KUKA KRL program: EPS_2_251806_MH03A_A_20260212042231.src

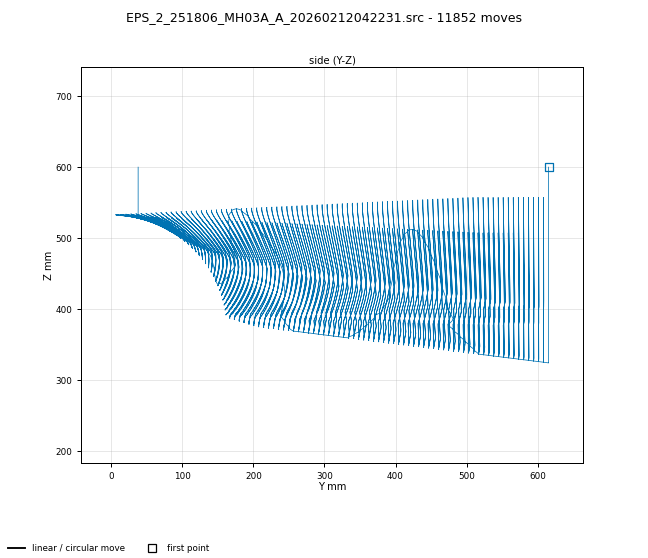
[picture p0: tool path of EPS_2_251806_MH03A_A_20260212042231.src, 11852 of 11854 moves have a stored position in this frame; points joined in program order, loops and branches not executed]
&ACCESS RVP
&REL 4
&COMMENT QRS 19112012
&PARAM EDITMASK = *
DEF PART()
EXT BAS (BAS_COMMAND :IN,REAL :IN )
INT I
BAS (#INITMOV,0 )

;KUKA QRS Post kuka4.cps  Date:22-06-2017 !

File_ID=3011

QRS_PRE_INIT()

;Init var - Until changes are made in qrs_pre_init
Outlet_Square_prg=0
Inlet_1_Square_prg=0
Inlet_2_Square_prg=0
Inlet_3_Square_prg=0
Inlet_4_Square_prg=0
Inlet_5_Square_prg=0

Outlet_1={X 0.000, Y 508.200, Z 408.000, B 0.000, E1 0.000 }
Inlet_1={X 0.000, Y 518.810, Z 382.000, B 0.000, E1 180.000 }
Outlet_1_type=299
Inlet_1_type=251
;QRS#1=Sidecore dimensions
;QRS#2=300-12" PVC SDR 35
;QRS#3=250-10" PVC SDR 35
;QRS#4=
;QRS#5=
;QRS#6=
;QRS#7=
;QRS#8=
;QRS#9=16M PSX
;QRS#10=14M PSX
;QRS#11=
;QRS#12=
;QRS#13=
;QRS#14=
;QRS#15=
;QRS#16=1220x127x838 2,75'
;QRS#17=EPS Height
;QRS#18=557,5
;QRS#19=*
;QRS#20= UPDATED VERSION 22-06-2017
;QRS#21=*
Outlet_Square=0150
Inlet_1_Square=0100
Inlet_2_Square=0
Inlet_3_Square=0
Inlet_4_Square=0
Inlet_5_Square=0
Mill_Square=1
Outlet_Square_Prg=206
Inlet_1_Square_prg=205

QRS_INIT()

$ADVANCE=5

; T1
PTP {E1 173.606,E2 173.606}
PTP {X 0,Y 615.511,A -85,B 0,C 180,E1 173.606,E2 173.606,E3 0,E4 0,E5 0,E6 0}
QRS_SPEED_INIT()
LIN {X 0,Y 615.511,Z 600,A -85,B 0,C 180,E1 173.606,E2 173.606,E3 0,E4 0,E5 0,E6 0} C_VEL
LIN {X 0,Y 615.511,Z 334.496,A -85,B 0,C 180,E1 173.606,E2 173.606} C_VEL
LIN {X 0,Y 615.511,Z 326.325,A -85,B 0,C 180,E1 173.606,E2 173.606} C_VEL
LIN {X 0,Y 615.495,Z 324.325,A -85,B 0,C 180,E1 173.42,E2 173.42} C_VEL
LIN {X 0,Y 615.489,Z 324.313,A -85,B 0,C 180,E1 170.801,E2 170.801} C_VEL
LIN {X 0,Y 615.492,Z 324.321,A -85,B 0,C 180,E1 168.139,E2 168.139} C_VEL
LIN {X 0,Y 615.481,Z 324.317,A -85,B 0,C 180,E1 165.451,E2 165.451} C_VEL
LIN {X 0,Y 615.493,Z 324.313,A -85,B 0,C 180,E1 162.73,E2 162.73} C_VEL
LIN {X 0,Y 615.493,Z 324.325,A -85,B 0,C 180,E1 159.967,E2 159.967} C_VEL
LIN {X 0,Y 615.481,Z 324.316,A -85,B 0,C 180,E1 157.155,E2 157.155} C_VEL
LIN {X 0,Y 615.475,Z 324.319,A -85,B 0,C 180,E1 154.435,E2 154.435} C_VEL
LIN {X 0,Y 615.485,Z 324.315,A -85,B 0,C 180,E1 152.085,E2 152.085} C_VEL
LIN {X 0,Y 615.5,Z 324.325,A -85,B 0,C 180,E1 149.84,E2 149.84} C_VEL
LIN {X 0,Y 615.474,Z 324.317,A -85,B 0,C 180,E1 147.542,E2 147.542} C_VEL
LIN {X 0,Y 615.491,Z 324.317,A -85,B 0,C 180,E1 145.185,E2 145.185} C_VEL
LIN {X 0,Y 615.479,Z 324.32,A -85,B 0,C 180,E1 142.757,E2 142.757} C_VEL
LIN {X 0,Y 615.495,Z 324.321,A -85,B 0,C 180,E1 139.911,E2 139.911} C_VEL
LIN {X 0,Y 615.485,Z 324.315,A -85,B 0,C 180,E1 136.953,E2 136.953} C_VEL
LIN {X 0,Y 615.481,Z 324.315,A -85,B 0,C 180,E1 133.997,E2 133.997} C_VEL
LIN {X 0,Y 615.488,Z 324.324,A -85,B 0,C 180,E1 131.474,E2 131.474} C_VEL
LIN {X 0,Y 615.478,Z 324.315,A -85,B 0,C 180,E1 128.905,E2 128.905} C_VEL
LIN {X 0,Y 615.496,Z 324.364,A -85,B 0,C 180,E1 128.172,E2 128.172} C_VEL
LIN {X 0,Y 615.485,Z 329.475,A -85,B 0,C 180,E1 125.616,E2 125.616} C_VEL
LIN {X 0,Y 615.491,Z 334.286,A -85,B 0,C 180,E1 123.236,E2 123.236} C_VEL
LIN {X 0,Y 615.478,Z 339.068,A -85,B 0,C 180,E1 120.92,E2 120.92} C_VEL
LIN {X 0,Y 615.491,Z 344.306,A -85,B 0,C 180,E1 118.45,E2 118.45} C_VEL
LIN {X 0,Y 615.498,Z 350.554,A -85,B 0,C 180,E1 115.57,E2 115.57} C_VEL
LIN {X 0,Y 615.49,Z 356.619,A -85,B 0,C 180,E1 112.845,E2 112.845} C_VEL
LIN {X 0,Y 615.479,Z 362.996,A -85,B 0,C 180,E1 110.033,E2 110.033} C_VEL
LIN {X 0,Y 615.497,Z 369.367,A -85,B 0,C 180,E1 107.27,E2 107.27} C_VEL
LIN {X 0,Y 615.482,Z 375.745,A -85,B 0,C 180,E1 104.549,E2 104.549} C_VEL
LIN {X 0,Y 615.484,Z 377.068,A -85,B 0,C 180,E1 103.99,E2 103.99} C_VEL
LIN {X 0,Y 615.487,Z 392.156,A -85,B 0,C 180,E1 103.706,E2 103.706} C_VEL
LIN {X 0,Y 615.478,Z 405.741,A -85,B 0,C 180,E1 103.328,E2 103.328} C_VEL
LIN {X 0,Y 615.488,Z 418.034,A -85,B 0,C 180,E1 102.865,E2 102.865} C_VEL
LIN {X 0,Y 615.479,Z 430.302,A -85,B 0,C 180,E1 102.279,E2 102.279} C_VEL
LIN {X 0,Y 615.498,Z 442.906,A -85,B 0,C 180,E1 101.527,E2 101.527} C_VEL
LIN {X 0,Y 615.498,Z 454.072,A -85,B 0,C 180,E1 100.709,E2 100.709} C_VEL
LIN {X 0,Y 615.499,Z 463.697,A -85,B 0,C 180,E1 99.862,E2 99.862} C_VEL
LIN {X 0,Y 615.497,Z 473.147,A -85,B 0,C 180,E1 98.867,E2 98.867} C_VEL
LIN {X 0,Y 615.497,Z 482.137,A -85,B 0,C 180,E1 97.71,E2 97.71} C_VEL
LIN {X 0,Y 615.496,Z 489.382,A -85,B 0,C 180,E1 96.557,E2 96.557} C_VEL
LIN {X 0,Y 615.494,Z 495.887,A -85,B 0,C 180,E1 95.241,E2 95.241} C_VEL
LIN {X 0,Y 615.496,Z 500.757,A -85,B 0,C 180,E1 93.928,E2 93.928} C_VEL
LIN {X 0,Y 615.496,Z 504.154,A -85,B 0,C 180,E1 92.618,E2 92.618} C_VEL
LIN {X 0,Y 615.493,Z 506.174,A -85,B 0,C 180,E1 91.309,E2 91.309} C_VEL
LIN {X 0,Y 615.494,Z 506.884,A -85,B 0,C 180,E1 90,E2 90} C_VEL
LIN {X 0,Y 615.49,Z 506.28,A -85,B 0,C 180,E1 88.691,E2 88.691} C_VEL
LIN {X 0,Y 615.493,Z 504.35,A -85,B 0,C 180,E1 87.382,E2 87.382} C_VEL
LIN {X 0,Y 615.496,Z 501.045,A -85,B 0,C 180,E1 86.071,E2 86.071} C_VEL
LIN {X 0,Y 615.496,Z 496.273,A -85,B 0,C 180,E1 84.759,E2 84.759} C_VEL
LIN {X 0,Y 615.495,Z 489.874,A -85,B 0,C 180,E1 83.443,E2 83.443} C_VEL
LIN {X 0,Y 615.496,Z 482.743,A -85,B 0,C 180,E1 82.289,E2 82.289} C_VEL
LIN {X 0,Y 615.497,Z 475.269,A -85,B 0,C 180,E1 81.298,E2 81.298} C_VEL
LIN {X 0,Y 615.496,Z 466.29,A -85,B 0,C 180,E1 80.304,E2 80.304} C_VEL
LIN {X 0,Y 615.499,Z 455.204,A -85,B 0,C 180,E1 79.291,E2 79.291} C_VEL
LIN {X 0,Y 615.498,Z 444.277,A -85,B 0,C 180,E1 78.473,E2 78.473} C_VEL
LIN {X 0,Y 615.479,Z 431.98,A -85,B 0,C 180,E1 77.721,E2 77.721} C_VEL
LIN {X 0,Y 615.488,Z 420.141,A -85,B 0,C 180,E1 77.134,E2 77.134} C_VEL
LIN {X 0,Y 615.478,Z 407.213,A -85,B 0,C 180,E1 76.63,E2 76.63} C_VEL
LIN {X 0,Y 615.489,Z 394.229,A -85,B 0,C 180,E1 76.252,E2 76.252} C_VEL
LIN {X 0,Y 615.482,Z 379.875,A -85,B 0,C 180,E1 75.972,E2 75.972} C_VEL
LIN {X 0,Y 615.479,Z 377.054,A -85,B 0,C 180,E1 75.914,E2 75.914} C_VEL
LIN {X 0,Y 615.489,Z 371.172,A -85,B 0,C 180,E1 73.413,E2 73.413} C_VEL
LIN {X 0,Y 615.495,Z 364.796,A -85,B 0,C 180,E1 70.662,E2 70.662} C_VEL
LIN {X 0,Y 615.478,Z 358.415,A -85,B 0,C 180,E1 67.863,E2 67.863} C_VEL
LIN {X 0,Y 615.478,Z 352.039,A -85,B 0,C 180,E1 65.008,E2 65.008} C_VEL
LIN {X 0,Y 615.476,Z 347.245,A -85,B 0,C 180,E1 62.822,E2 62.822} C_VEL
LIN {X 0,Y 615.495,Z 341.623,A -85,B 0,C 180,E1 60.205,E2 60.205} C_VEL
LIN {X 0,Y 615.493,Z 336.065,A -85,B 0,C 180,E1 57.542,E2 57.542} C_VEL
LIN {X 0,Y 615.495,Z 331.272,A -85,B 0,C 180,E1 55.185,E2 55.185} C_VEL
LIN {X 0,Y 615.487,Z 326.404,A -85,B 0,C 180,E1 52.757,E2 52.757} C_VEL
LIN {X 0,Y 615.487,Z 324.319,A -85,B 0,C 180,E1 51.619,E2 51.619} C_VEL
LIN {X 0,Y 615.484,Z 324.319,A -85,B 0,C 180,E1 48.906,E2 48.906} C_VEL
LIN {X 0,Y 615.499,Z 324.321,A -85,B 0,C 180,E1 46.756,E2 46.756} C_VEL
LIN {X 0,Y 615.484,Z 324.317,A -85,B 0,C 180,E1 43.996,E2 43.996} C_VEL
LIN {X 0,Y 615.482,Z 324.314,A -85,B 0,C 180,E1 41.093,E2 41.093} C_VEL
LIN {X 0,Y 615.492,Z 324.316,A -85,B 0,C 180,E1 38.904,E2 38.904} C_VEL
LIN {X 0,Y 615.478,Z 324.32,A -85,B 0,C 180,E1 36.426,E2 36.426} C_VEL
LIN {X 0,Y 615.497,Z 324.323,A -85,B 0,C 180,E1 33.535,E2 33.535} C_VEL
LIN {X 0,Y 615.488,Z 324.313,A -85,B 0,C 180,E1 30.92,E2 30.92} C_VEL
LIN {X 0,Y 615.498,Z 324.324,A -85,B 0,C 180,E1 28.451,E2 28.451} C_VEL
LIN {X 0,Y 615.478,Z 324.316,A -85,B 0,C 180,E1 25.716,E2 25.716} C_VEL
LIN {X 0,Y 615.485,Z 324.323,A -85,B 0,C 180,E1 23.557,E2 23.557} C_VEL
LIN {X 0,Y 615.493,Z 324.319,A -85,B 0,C 180,E1 21.432,E2 21.432} C_VEL
LIN {X 0,Y 615.482,Z 324.321,A -85,B 0,C 180,E1 18.601,E2 18.601} C_VEL
LIN {X 0,Y 615.478,Z 324.315,A -85,B 0,C 180,E1 15.906,E2 15.906} C_VEL
LIN {X 0,Y 615.493,Z 324.324,A -85,B 0,C 180,E1 13.201,E2 13.201} C_VEL
LIN {X 0,Y 615.486,Z 324.315,A -85,B 0,C 180,E1 10.527,E2 10.527} C_VEL
LIN {X 0,Y 615.479,Z 324.319,A -85,B 0,C 180,E1 7.876,E2 7.876} C_VEL
LIN {X 0,Y 615.494,Z 324.316,A -85,B 0,C 180,E1 5.241,E2 5.241} C_VEL
LIN {X 0,Y 615.488,Z 324.314,A -85,B 0,C 180,E1 2.618,E2 2.618} C_VEL
LIN {X 0,Y 615.488,Z 324.323,A -85,B 0,C 180,E1 0,E2 0} C_VEL
LIN {X 0,Y 615.488,Z 324.313,A -85,B 0,C 180,E1 -2.618,E2 -2.618} C_VEL
LIN {X 0,Y 615.496,Z 324.324,A -85,B 0,C 180,E1 -5.241,E2 -5.241} C_VEL
LIN {X 0,Y 615.478,Z 324.316,A -85,B 0,C 180,E1 -7.876,E2 -7.876} C_VEL
LIN {X 0,Y 615.486,Z 324.32,A -85,B 0,C 180,E1 -10.527,E2 -10.527} C_VEL
LIN {X 0,Y 615.494,Z 324.316,A -85,B 0,C 180,E1 -13.201,E2 -13.201} C_VEL
LIN {X 0,Y 615.478,Z 324.316,A -85,B 0,C 180,E1 -15.905,E2 -15.905} C_VEL
LIN {X 0,Y 615.493,Z 324.326,A -85,B 0,C 180,E1 -18.646,E2 -18.646} C_VEL
LIN {X 0,Y 615.479,Z 324.317,A -85,B 0,C 180,E1 -21.432,E2 -21.432} C_VEL
LIN {X 0,Y 615.487,Z 324.314,A -85,B 0,C 180,E1 -24.272,E2 -24.272} C_VEL
LIN {X 0,Y 615.49,Z 324.323,A -85,B 0,C 180,E1 -27.177,E2 -27.177} C_VEL
LIN {X 0,Y 615.485,Z 324.315,A -85,B 0,C 180,E1 -29.793,E2 -29.793} C_VEL
LIN {X 0,Y 615.477,Z 324.32,A -85,B 0,C 180,E1 -32.458,E2 -32.458} C_VEL
LIN {X 0,Y 615.491,Z 324.313,A -85,B 0,C 180,E1 -34.815,E2 -34.815} C_VEL
LIN {X 0,Y 615.492,Z 324.323,A -85,B 0,C 180,E1 -37.242,E2 -37.242} C_VEL
LIN {X 0,Y 615.491,Z 324.317,A -85,B 0,C 180,E1 -40.089,E2 -40.089} C_VEL
LIN {X 0,Y 615.483,Z 324.314,A -85,B 0,C 180,E1 -43.046,E2 -43.046} C_VEL
LIN {X 0,Y 615.482,Z 324.317,A -85,B 0,C 180,E1 -46.003,E2 -46.003} C_VEL
LIN {X 0,Y 615.488,Z 324.318,A -85,B 0,C 180,E1 -48.526,E2 -48.526} C_VEL
LIN {X 0,Y 615.478,Z 324.317,A -85,B 0,C 180,E1 -51.094,E2 -51.094} C_VEL
LIN {X 0,Y 615.489,Z 324.318,A -85,B 0,C 180,E1 -53.575,E2 -53.575} C_VEL
LIN {X 0,Y 615.479,Z 324.469,A -85,B 0,C 180,E1 -55.242,E2 -55.242} C_VEL
LIN {X 0,Y 615.492,Z 334.986,A -85,B 0,C 180,E1 -57.992,E2 -57.992} C_VEL
LIN {X 0,Y 615.492,Z 345.267,A -85,B 0,C 180,E1 -60.594,E2 -60.594} C_VEL
LIN {X 0,Y 615.487,Z 356.058,A -85,B 0,C 180,E1 -63.257,E2 -63.257} C_VEL
LIN {X 0,Y 615.478,Z 367.411,A -85,B 0,C 180,E1 -65.994,E2 -65.994} C_VEL
LIN {X 0,Y 615.481,Z 378.295,A -85,B 0,C 180,E1 -68.568,E2 -68.568} C_VEL
LIN {X 0,Y 615.489,Z 390.473,A -85,B 0,C 180,E1 -71.395,E2 -71.395} C_VEL
LIN {X 0,Y 615.488,Z 400.106,A -85,B 0,C 180,E1 -73.601,E2 -73.601} C_VEL
LIN {X 0,Y 615.493,Z 417.365,A -85,B 0,C 180,E1 -73.865,E2 -73.865} C_VEL
LIN {X 0,Y 615.497,Z 432.278,A -85,B 0,C 180,E1 -74.222,E2 -74.222} C_VEL
LIN {X 0,Y 615.478,Z 446.42,A -85,B 0,C 180,E1 -74.689,E2 -74.689} C_VEL
LIN {X 0,Y 615.496,Z 460.354,A -85,B 0,C 180,E1 -75.282,E2 -75.282} C_VEL
LIN {X 0,Y 615.499,Z 473.673,A -85,B 0,C 180,E1 -75.986,E2 -75.986} C_VEL
LIN {X 0,Y 615.498,Z 486.312,A -85,B 0,C 180,E1 -76.799,E2 -76.799} C_VEL
LIN {X 0,Y 615.496,Z 497.291,A -85,B 0,C 180,E1 -77.637,E2 -77.637} C_VEL
LIN {X 0,Y 615.497,Z 508.352,A -85,B 0,C 180,E1 -78.64,E2 -78.64} C_VEL
LIN {X 0,Y 615.496,Z 519.068,A -85,B 0,C 180,E1 -79.806,E2 -79.806} C_VEL
LIN {X 0,Y 615.495,Z 527.987,A -85,B 0,C 180,E1 -80.967,E2 -80.967} C_VEL
LIN {X 0,Y 615.492,Z 535.392,A -85,B 0,C 180,E1 -82.124,E2 -82.124} C_VEL
LIN {X 0,Y 615.491,Z 542.272,A -85,B 0,C 180,E1 -83.443,E2 -83.443} C_VEL
LIN {X 0,Y 615.491,Z 547.666,A -85,B 0,C 180,E1 -84.759,E2 -84.759} C_VEL
LIN {X 0,Y 615.491,Z 551.741,A -85,B 0,C 180,E1 -86.071,E2 -86.071} C_VEL
LIN {X 0,Y 615.496,Z 554.599,A -85,B 0,C 180,E1 -87.382,E2 -87.382} C_VEL
LIN {X 0,Y 615.493,Z 556.306,A -85,B 0,C 180,E1 -88.691,E2 -88.691} C_VEL
LIN {X 0,Y 615.491,Z 556.889,A -85,B 0,C 180,E1 -90,E2 -90} C_VEL
LIN {X 0,Y 615.493,Z 556.307,A -85,B 0,C 180,E1 -91.309,E2 -91.309} C_VEL
LIN {X 0,Y 615.496,Z 554.599,A -85,B 0,C 180,E1 -92.618,E2 -92.618} C_VEL
LIN {X 0,Y 615.491,Z 551.741,A -85,B 0,C 180,E1 -93.928,E2 -93.928} C_VEL
LIN {X 0,Y 615.491,Z 547.666,A -85,B 0,C 180,E1 -95.241,E2 -95.241} C_VEL
LIN {X 0,Y 615.491,Z 542.153,A -85,B 0,C 180,E1 -96.581,E2 -96.581} C_VEL
LIN {X 0,Y 615.492,Z 535.393,A -85,B 0,C 180,E1 -97.876,E2 -97.876} C_VEL
LIN {X 0,Y 615.495,Z 526.809,A -85,B 0,C 180,E1 -99.199,E2 -99.199} C_VEL
LIN {X 0,Y 615.494,Z 517.667,A -85,B 0,C 180,E1 -100.361,E2 -100.361} C_VEL
LIN {X 0,Y 615.497,Z 508.353,A -85,B 0,C 180,E1 -101.36,E2 -101.36} C_VEL
LIN {X 0,Y 615.496,Z 497.292,A -85,B 0,C 180,E1 -102.363,E2 -102.363} C_VEL
LIN {X 0,Y 615.498,Z 485.152,A -85,B 0,C 180,E1 -103.285,E2 -103.285} C_VEL
LIN {X 0,Y 615.498,Z 472.405,A -85,B 0,C 180,E1 -104.09,E2 -104.09} C_VEL
LIN {X 0,Y 615.496,Z 458.609,A -85,B 0,C 180,E1 -104.803,E2 -104.803} C_VEL
LIN {X 0,Y 615.48,Z 444.181,A -85,B 0,C 180,E1 -105.396,E2 -105.396} C_VEL
LIN {X 0,Y 615.496,Z 429.246,A -85,B 0,C 180,E1 -105.863,E2 -105.863} C_VEL
LIN {X 0,Y 615.491,Z 413.842,A -85,B 0,C 180,E1 -106.201,E2 -106.201} C_VEL
LIN {X 0,Y 615.488,Z 400.106,A -85,B 0,C 180,E1 -106.399,E2 -106.399} C_VEL
LIN {X 0,Y 615.484,Z 388.794,A -85,B 0,C 180,E1 -108.992,E2 -108.992} C_VEL
LIN {X 0,Y 615.489,Z 376.797,A -85,B 0,C 180,E1 -111.784,E2 -111.784} C_VEL
LIN {X 0,Y 615.493,Z 364.791,A -85,B 0,C 180,E1 -114.631,E2 -114.631} C_VEL
LIN {X 0,Y 615.494,Z 352.781,A -85,B 0,C 180,E1 -117.545,E2 -117.545} C_VEL
LIN {X 0,Y 615.496,Z 340.758,A -85,B 0,C 180,E1 -120.539,E2 -120.539} C_VEL
LIN {X 0,Y 615.485,Z 330.231,A -85,B 0,C 180,E1 -123.237,E2 -123.237} C_VEL
LIN {X 0,Y 615.478,Z 324.319,A -85,B 0,C 180,E1 -124.816,E2 -124.816} C_VEL
LIN {X 0,Y 615.486,Z 324.315,A -85,B 0,C 180,E1 -127.243,E2 -127.243} C_VEL
LIN {X 0,Y 615.484,Z 324.315,A -85,B 0,C 180,E1 -130.089,E2 -130.089} C_VEL
LIN {X 0,Y 615.498,Z 324.314,A -85,B 0,C 180,E1 -132.353,E2 -132.353} C_VEL
LIN {X 0,Y 615.48,Z 324.316,A -85,B 0,C 180,E1 -135.07,E2 -135.07} C_VEL
LIN {X 0,Y 615.499,Z 324.324,A -85,B 0,C 180,E1 -137.919,E2 -137.919} C_VEL
LIN {X 0,Y 615.491,Z 324.313,A -85,B 0,C 180,E1 -140.25,E2 -140.25} C_VEL
LIN {X 0,Y 615.493,Z 324.322,A -85,B 0,C 180,E1 -143.063,E2 -143.063} C_VEL
LIN {X 0,Y 615.489,Z 324.319,A -85,B 0,C 180,E1 -145.978,E2 -145.978} C_VEL
LIN {X 0,Y 615.484,Z 324.314,A -85,B 0,C 180,E1 -148.915,E2 -148.915} C_VEL
LIN {X 0,Y 615.487,Z 324.321,A -85,B 0,C 180,E1 -151.551,E2 -151.551} C_VEL
LIN {X 0,Y 615.487,Z 324.317,A -85,B 0,C 180,E1 -154.284,E2 -154.284} C_VEL
LIN {X 0,Y 615.481,Z 324.314,A -85,B 0,C 180,E1 -157.155,E2 -157.155} C_VEL
LIN {X 0,Y 615.49,Z 324.32,A -85,B 0,C 180,E1 -159.967,E2 -159.967} C_VEL
LIN {X 0,Y 615.493,Z 324.317,A -85,B 0,C 180,E1 -162.73,E2 -162.73} C_VEL
LIN {X 0,Y 615.482,Z 324.315,A -85,B 0,C 180,E1 -165.451,E2 -165.451} C_VEL
LIN {X 0,Y 615.493,Z 324.326,A -85,B 0,C 180,E1 -168.139,E2 -168.139} C_VEL
LIN {X 0,Y 615.489,Z 324.313,A -85,B 0,C 180,E1 -170.801,E2 -170.801} C_VEL
LIN {X 0,Y 615.496,Z 324.318,A -85,B 0,C 180,E1 -173.444,E2 -173.444} C_VEL
LIN {X 0,Y 615.479,Z 324.318,A -85,B 0,C 180,E1 -176.072,E2 -176.072} C_VEL
LIN {X 0,Y 615.487,Z 324.316,A -85,B 0,C 180,E1 -178.692,E2 -178.692} C_VEL
LIN {X 0,Y 615.487,Z 324.32,A -85,B 0,C 180,E1 -181.309,E2 -181.309} C_VEL
LIN {X 0,Y 615.477,Z 324.316,A -85,B 0,C 180,E1 -183.929,E2 -183.929} C_VEL
LIN {X 0,Y 615.495,Z 324.325,A -85,B 0,C 180,E1 -186.58,E2 -186.58} C_VEL
LIN {X 0,Y 614.815,Z 324.462,A -85,B 0,C 180,E1 -187.126,E2 -187.126} C_VEL
LIN {X 0,Y 611.977,Z 324.88,A -85,B 0,C 180,E1 -188.012,E2 -188.012} C_VEL
LIN {X 0,Y 609.586,Z 325.186,A -85,B 0,C 180,E1 -188.724,E2 -188.724} C_VEL
LIN {X 0,Y 608.552,Z 325.304,A -85,B 0,C 180,E1 -189.274,E2 -189.274} C_VEL
LIN {X 0,Y 608.463,Z 325.315,A -85,B 0,C 180,E1 -189.46,E2 -189.46} C_VEL
LIN {X 0,Y 608.466,Z 325.317,A -85,B 0,C 180,E1 -192,E2 -192} C_VEL
LIN {X 0,Y 608.474,Z 325.316,A -85,B 0,C 180,E1 -194.721,E2 -194.721} C_VEL
LIN {X 0,Y 608.456,Z 325.315,A -85,B 0,C 180,E1 -197.477,E2 -197.477} C_VEL
LIN {X 0,Y 608.462,Z 325.319,A -85,B 0,C 180,E1 -200.274,E2 -200.274} C_VEL
LIN {X 0,Y 608.464,Z 325.314,A -85,B 0,C 180,E1 -202.476,E2 -202.476} C_VEL
LIN {X 0,Y 608.457,Z 325.316,A -85,B 0,C 180,E1 -204.571,E2 -204.571} C_VEL
LIN {X 0,Y 608.485,Z 325.313,A -85,B 0,C 180,E1 -207.207,E2 -207.207} C_VEL
LIN {X 0,Y 608.471,Z 325.318,A -85,B 0,C 180,E1 -209.971,E2 -209.971} C_VEL
LIN {X 0,Y 608.457,Z 325.315,A -85,B 0,C 180,E1 -212.88,E2 -212.88} C_VEL
LIN {X 0,Y 608.443,Z 325.323,A -85,B 0,C 180,E1 -215.278,E2 -215.278} C_VEL
LIN {X 0,Y 608.467,Z 325.314,A -85,B 0,C 180,E1 -217.747,E2 -217.747} C_VEL
LIN {X 0,Y 608.458,Z 325.321,A -85,B 0,C 180,E1 -220.329,E2 -220.329} C_VEL
LIN {X 0,Y 608.451,Z 325.316,A -85,B 0,C 180,E1 -222.96,E2 -222.96} C_VEL
LIN {X 0,Y 608.46,Z 325.316,A -85,B 0,C 180,E1 -225.736,E2 -225.736} C_VEL
LIN {X 0,Y 608.463,Z 325.322,A -85,B 0,C 180,E1 -228.658,E2 -228.658} C_VEL
LIN {X 0,Y 608.483,Z 325.333,A -85,B 0,C 180,E1 -231.758,E2 -231.758} C_VEL
LIN {X 0,Y 608.48,Z 331.224,A -85,B 0,C 180,E1 -234.725,E2 -234.725} C_VEL
LIN {X 0,Y 608.467,Z 336.749,A -85,B 0,C 180,E1 -237.477,E2 -237.477} C_VEL
LIN {X 0,Y 608.481,Z 342.43,A -85,B 0,C 180,E1 -240.221,E2 -240.221} C_VEL
LIN {X 0,Y 608.435,Z 348.844,A -85,B 0,C 180,E1 -243.225,E2 -243.225} C_VEL
LIN {X 0,Y 608.452,Z 354.592,A -85,B 0,C 180,E1 -245.853,E2 -245.853} C_VEL
LIN {X 0,Y 608.443,Z 360.069,A -85,B 0,C 180,E1 -248.307,E2 -248.307} C_VEL
LIN {X 0,Y 608.43,Z 366.867,A -85,B 0,C 180,E1 -251.296,E2 -251.296} C_VEL
LIN {X 0,Y 608.442,Z 372.899,A -85,B 0,C 180,E1 -253.906,E2 -253.906} C_VEL
LIN {X 0,Y 608.43,Z 377.462,A -85,B 0,C 180,E1 -255.856,E2 -255.856} C_VEL
LIN {X 0,Y 608.599,Z 393.096,A -85,B 0,C 180,E1 -256.157,E2 -256.157} C_VEL
LIN {X 0,Y 608.553,Z 407.065,A -85,B 0,C 180,E1 -256.561,E2 -256.561} C_VEL
LIN {X 0,Y 608.54,Z 420.049,A -85,B 0,C 180,E1 -257.07,E2 -257.07} C_VEL
LIN {X 0,Y 608.529,Z 431.94,A -85,B 0,C 180,E1 -257.663,E2 -257.663} C_VEL
LIN {X 0,Y 608.509,Z 444.298,A -85,B 0,C 180,E1 -258.424,E2 -258.424} C_VEL
LIN {X 0,Y 608.501,Z 456.473,A -85,B 0,C 180,E1 -259.351,E2 -259.351} C_VEL
LIN {X 0,Y 608.469,Z 467.272,A -85,B 0,C 180,E1 -260.359,E2 -260.359} C_VEL
LIN {X 0,Y 608.47,Z 476.191,A -85,B 0,C 180,E1 -261.364,E2 -261.364} C_VEL
LIN {X 0,Y 608.47,Z 484.736,A -85,B 0,C 180,E1 -262.534,E2 -262.534} C_VEL
LIN {X 0,Y 608.443,Z 492.325,A -85,B 0,C 180,E1 -263.831,E2 -263.831} C_VEL
LIN {X 0,Y 608.435,Z 497.788,A -85,B 0,C 180,E1 -265.03,E2 -265.03} C_VEL
LIN {X 0,Y 608.434,Z 501.298,A -85,B 0,C 180,E1 -266.026,E2 -266.026} C_VEL
LIN {X 0,Y 608.424,Z 504.734,A -85,B 0,C 180,E1 -267.352,E2 -267.352} C_VEL
LIN {X 0,Y 608.446,Z 506.777,A -85,B 0,C 180,E1 -268.676,E2 -268.676} C_VEL
LIN {X 0,Y 608.434,Z 507.495,A -85,B 0,C 180,E1 -270,E2 -270} C_VEL
LIN {X 0,Y 608.443,Z 506.882,A -85,B 0,C 180,E1 -271.324,E2 -271.324} C_VEL
LIN {X 0,Y 608.421,Z 504.928,A -85,B 0,C 180,E1 -272.648,E2 -272.648} C_VEL
LIN {X 0,Y 608.434,Z 501.584,A -85,B 0,C 180,E1 -273.974,E2 -273.974} C_VEL
LIN {X 0,Y 608.44,Z 496.759,A -85,B 0,C 180,E1 -275.302,E2 -275.302} C_VEL
LIN {X 0,Y 608.443,Z 490.472,A -85,B 0,C 180,E1 -276.601,E2 -276.601} C_VEL
LIN {X 0,Y 608.453,Z 483.098,A -85,B 0,C 180,E1 -277.8,E2 -277.8} C_VEL
LIN {X 0,Y 608.476,Z 475.561,A -85,B 0,C 180,E1 -278.803,E2 -278.803} C_VEL
LIN {X 0,Y 608.488,Z 466.516,A -85,B 0,C 180,E1 -279.809,E2 -279.809} C_VEL
LIN {X 0,Y 608.507,Z 455.723,A -85,B 0,C 180,E1 -280.804,E2 -280.804} C_VEL
LIN {X 0,Y 608.524,Z 444.379,A -85,B 0,C 180,E1 -281.661,E2 -281.661} C_VEL
LIN {X 0,Y 608.53,Z 432.036,A -85,B 0,C 180,E1 -282.422,E2 -282.422} C_VEL
LIN {X 0,Y 608.551,Z 420.165,A -85,B 0,C 180,E1 -283.015,E2 -283.015} C_VEL
LIN {X 0,Y 608.566,Z 407.211,A -85,B 0,C 180,E1 -283.524,E2 -283.524} C_VEL
LIN {X 0,Y 608.592,Z 393.013,A -85,B 0,C 180,E1 -283.935,E2 -283.935} C_VEL
LIN {X 0,Y 608.541,Z 378.307,A -85,B 0,C 180,E1 -284.213,E2 -284.213} C_VEL
LIN {X 0,Y 608.417,Z 377.471,A -85,B 0,C 180,E1 -284.231,E2 -284.231} C_VEL
LIN {X 0,Y 608.447,Z 371.504,A -85,B 0,C 180,E1 -286.784,E2 -286.784} C_VEL
LIN {X 0,Y 608.436,Z 365.086,A -85,B 0,C 180,E1 -289.571,E2 -289.571} C_VEL
LIN {X 0,Y 608.432,Z 358.527,A -85,B 0,C 180,E1 -292.47,E2 -292.47} C_VEL
LIN {X 0,Y 608.436,Z 352.248,A -85,B 0,C 180,E1 -295.302,E2 -295.302} C_VEL
LIN {X 0,Y 608.448,Z 345.829,A -85,B 0,C 180,E1 -298.267,E2 -298.267} C_VEL
LIN {X 0,Y 608.446,Z 341.014,A -85,B 0,C 180,E1 -300.547,E2 -300.547} C_VEL
LIN {X 0,Y 608.464,Z 336.222,A -85,B 0,C 180,E1 -302.88,E2 -302.88} C_VEL
LIN {X 0,Y 608.45,Z 331.386,A -85,B 0,C 180,E1 -305.278,E2 -305.278} C_VEL
LIN {X 0,Y 608.492,Z 325.43,A -85,B 0,C 180,E1 -308.281,E2 -308.281} C_VEL
LIN {X 0,Y 608.467,Z 325.32,A -85,B 0,C 180,E1 -311.342,E2 -311.342} C_VEL
LIN {X 0,Y 608.461,Z 325.315,A -85,B 0,C 180,E1 -314.264,E2 -314.264} C_VEL
LIN {X 0,Y 608.454,Z 325.316,A -85,B 0,C 180,E1 -317.04,E2 -317.04} C_VEL
LIN {X 0,Y 608.459,Z 325.32,A -85,B 0,C 180,E1 -319.697,E2 -319.697} C_VEL
LIN {X 0,Y 608.47,Z 325.313,A -85,B 0,C 180,E1 -322.254,E2 -322.254} C_VEL
LIN {X 0,Y 608.455,Z 325.319,A -85,B 0,C 180,E1 -325.095,E2 -325.095} C_VEL
LIN {X 0,Y 608.452,Z 325.315,A -85,B 0,C 180,E1 -327.48,E2 -327.48} C_VEL
LIN {X 0,Y 608.47,Z 325.316,A -85,B 0,C 180,E1 -330.22,E2 -330.22} C_VEL
LIN {X 0,Y 608.485,Z 325.313,A -85,B 0,C 180,E1 -332.793,E2 -332.793} C_VEL
LIN {X 0,Y 608.483,Z 325.312,A -85,B 0,C 180,E1 -335.848,E2 -335.848} C_VEL
LIN {X 0,Y 608.476,Z 325.32,A -85,B 0,C 180,E1 -338.309,E2 -338.309} C_VEL
LIN {X 0,Y 608.471,Z 325.315,A -85,B 0,C 180,E1 -341.286,E2 -341.286} C_VEL
LIN {X 0,Y 608.46,Z 325.315,A -85,B 0,C 180,E1 -343.906,E2 -343.906} C_VEL
LIN {X 0,Y 608.467,Z 325.32,A -85,B 0,C 180,E1 -346.644,E2 -346.644} C_VEL
LIN {X 0,Y 608.462,Z 325.314,A -85,B 0,C 180,E1 -349.35,E2 -349.35} C_VEL
LIN {X 0,Y 608.474,Z 325.316,A -85,B 0,C 180,E1 -352.033,E2 -352.033} C_VEL
LIN {X 0,Y 608.472,Z 325.315,A -85,B 0,C 180,E1 -354.698,E2 -354.698} C_VEL
LIN {X 0,Y 608.48,Z 325.313,A -85,B 0,C 180,E1 -357.352,E2 -357.352} C_VEL
LIN {X 0,Y 608.479,Z 325.318,A -85,B 0,C 180,E1 -360,E2 -360} C_VEL
LIN {X 0,Y 608.479,Z 325.312,A -85,B 0,C 180,E1 -362.648,E2 -362.648} C_VEL
LIN {X 0,Y 608.474,Z 325.319,A -85,B 0,C 180,E1 -365.302,E2 -365.302} C_VEL
LIN {X 0,Y 608.473,Z 325.313,A -85,B 0,C 180,E1 -367.967,E2 -367.967} C_VEL
LIN {X 0,Y 608.462,Z 325.316,A -85,B 0,C 180,E1 -370.65,E2 -370.65} C_VEL
LIN {X 0,Y 608.47,Z 325.318,A -85,B 0,C 180,E1 -373.356,E2 -373.356} C_VEL
LIN {X 0,Y 608.458,Z 325.315,A -85,B 0,C 180,E1 -376.094,E2 -376.094} C_VEL
LIN {X 0,Y 608.462,Z 325.318,A -85,B 0,C 180,E1 -378.869,E2 -378.869} C_VEL
LIN {X 0,Y 608.469,Z 325.317,A -85,B 0,C 180,E1 -381.691,E2 -381.691} C_VEL
LIN {X 0,Y 608.457,Z 325.315,A -85,B 0,C 180,E1 -384.571,E2 -384.571} C_VEL
LIN {X 0,Y 608.485,Z 325.316,A -85,B 0,C 180,E1 -387.207,E2 -387.207} C_VEL
LIN {X 0,Y 608.47,Z 325.315,A -85,B 0,C 180,E1 -389.971,E2 -389.971} C_VEL
LIN {X 0,Y 608.453,Z 325.315,A -85,B 0,C 180,E1 -392.88,E2 -392.88} C_VEL
LIN {X 0,Y 608.451,Z 325.321,A -85,B 0,C 180,E1 -395.277,E2 -395.277} C_VEL
LIN {X 0,Y 608.471,Z 325.314,A -85,B 0,C 180,E1 -397.746,E2 -397.746} C_VEL
LIN {X 0,Y 608.458,Z 325.32,A -85,B 0,C 180,E1 -400.329,E2 -400.329} C_VEL
LIN {X 0,Y 608.449,Z 325.316,A -85,B 0,C 180,E1 -402.96,E2 -402.96} C_VEL
LIN {X 0,Y 608.459,Z 325.319,A -85,B 0,C 180,E1 -405.736,E2 -405.736} C_VEL
LIN {X 0,Y 608.465,Z 325.318,A -85,B 0,C 180,E1 -408.657,E2 -408.657} C_VEL
LIN {X 0,Y 608.471,Z 325.315,A -85,B 0,C 180,E1 -411.759,E2 -411.759} C_VEL
LIN {X 0,Y 608.447,Z 325.324,A -85,B 0,C 180,E1 -413.954,E2 -413.954} C_VEL
LIN {X 0,Y 608.483,Z 325.503,A -85,B 0,C 180,E1 -415.049,E2 -415.049} C_VEL
LIN {X 0,Y 608.544,Z 333.241,A -85,B 0,C 180,E1 -417.125,E2 -417.125} C_VEL
LIN {X 0,Y 608.555,Z 343.531,A -85,B 0,C 180,E1 -419.781,E2 -419.781} C_VEL
LIN {X 0,Y 608.534,Z 354.309,A -85,B 0,C 180,E1 -422.486,E2 -422.486} C_VEL
LIN {X 0,Y 608.489,Z 364.843,A -85,B 0,C 180,E1 -425.066,E2 -425.066} C_VEL
LIN {X 0,Y 608.479,Z 375.378,A -85,B 0,C 180,E1 -427.595,E2 -427.595} C_VEL
LIN {X 0,Y 608.482,Z 387.417,A -85,B 0,C 180,E1 -430.43,E2 -430.43} C_VEL
LIN {X 0,Y 608.461,Z 399.909,A -85,B 0,C 180,E1 -433.32,E2 -433.32} C_VEL
LIN {X 0,Y 608.461,Z 400.31,A -85,B 0,C 180,E1 -433.412,E2 -433.412} C_VEL
LIN {X 0,Y 608.678,Z 412.209,A -85,B 0,C 180,E1 -433.582,E2 -433.582} C_VEL
LIN {X 0,Y 608.656,Z 427.704,A -85,B 0,C 180,E1 -433.911,E2 -433.911} C_VEL
LIN {X 0,Y 608.629,Z 443.044,A -85,B 0,C 180,E1 -434.383,E2 -434.383} C_VEL
LIN {X 0,Y 608.615,Z 456.751,A -85,B 0,C 180,E1 -434.94,E2 -434.94} C_VEL
LIN {X 0,Y 608.582,Z 470.233,A -85,B 0,C 180,E1 -435.624,E2 -435.624} C_VEL
LIN {X 0,Y 608.554,Z 482.661,A -85,B 0,C 180,E1 -436.39,E2 -436.39} C_VEL
LIN {X 0,Y 608.528,Z 495.281,A -85,B 0,C 180,E1 -437.324,E2 -437.324} C_VEL
LIN {X 0,Y 608.496,Z 506.746,A -85,B 0,C 180,E1 -438.339,E2 -438.339} C_VEL
LIN {X 0,Y 608.477,Z 516.387,A -85,B 0,C 180,E1 -439.35,E2 -439.35} C_VEL
LIN {X 0,Y 608.476,Z 525.853,A -85,B 0,C 180,E1 -440.526,E2 -440.526} C_VEL
LIN {X 0,Y 608.456,Z 533.728,A -85,B 0,C 180,E1 -441.698,E2 -441.698} C_VEL
LIN {X 0,Y 608.441,Z 541.087,A -85,B 0,C 180,E1 -443.034,E2 -443.034} C_VEL
LIN {X 0,Y 608.45,Z 546.923,A -85,B 0,C 180,E1 -444.365,E2 -444.365} C_VEL
LIN {X 0,Y 608.427,Z 550.382,A -85,B 0,C 180,E1 -445.362,E2 -445.362} C_VEL
LIN {X 0,Y 608.421,Z 553.885,A -85,B 0,C 180,E1 -446.689,E2 -446.689} C_VEL
LIN {X 0,Y 608.444,Z 556.191,A -85,B 0,C 180,E1 -448.014,E2 -448.014} C_VEL
LIN {X 0,Y 608.436,Z 557.351,A -85,B 0,C 180,E1 -449.338,E2 -449.338} C_VEL
LIN {X 0,Y 608.436,Z 557.351,A -85,B 0,C 180,E1 -450.662,E2 -450.662} C_VEL
LIN {X 0,Y 608.444,Z 556.191,A -85,B 0,C 180,E1 -451.986,E2 -451.986} C_VEL
LIN {X 0,Y 608.421,Z 553.886,A -85,B 0,C 180,E1 -453.311,E2 -453.311} C_VEL
LIN {X 0,Y 608.427,Z 550.383,A -85,B 0,C 180,E1 -454.638,E2 -454.638} C_VEL
LIN {X 0,Y 608.437,Z 545.608,A -85,B 0,C 180,E1 -455.967,E2 -455.967} C_VEL
LIN {X 0,Y 608.457,Z 539.426,A -85,B 0,C 180,E1 -457.299,E2 -457.299} C_VEL
LIN {X 0,Y 608.468,Z 531.654,A -85,B 0,C 180,E1 -458.636,E2 -458.636} C_VEL
LIN {X 0,Y 608.471,Z 523.37,A -85,B 0,C 180,E1 -459.809,E2 -459.809} C_VEL
LIN {X 0,Y 608.493,Z 512.648,A -85,B 0,C 180,E1 -461.063,E2 -461.063} C_VEL
LIN {X 0,Y 608.522,Z 501.274,A -85,B 0,C 180,E1 -462.168,E2 -462.168} C_VEL
LIN {X 0,Y 608.547,Z 489.853,A -85,B 0,C 180,E1 -463.1,E2 -463.1} C_VEL
LIN {X 0,Y 608.563,Z 477.445,A -85,B 0,C 180,E1 -463.95,E2 -463.95} C_VEL
LIN {X 0,Y 608.602,Z 463.857,A -85,B 0,C 180,E1 -464.717,E2 -464.717} C_VEL
LIN {X 0,Y 608.599,Z 449.789,A -85,B 0,C 180,E1 -465.36,E2 -465.36} C_VEL
LIN {X 0,Y 608.661,Z 434.562,A -85,B 0,C 180,E1 -465.895,E2 -465.895} C_VEL
LIN {X 0,Y 608.69,Z 419.966,A -85,B 0,C 180,E1 -466.271,E2 -466.271} C_VEL
LIN {X 0,Y 608.689,Z 403.976,A -85,B 0,C 180,E1 -466.535,E2 -466.535} C_VEL
LIN {X 0,Y 608.458,Z 400.24,A -85,B 0,C 180,E1 -466.604,E2 -466.604} C_VEL
LIN {X 0,Y 608.46,Z 388.922,A -85,B 0,C 180,E1 -469.22,E2 -469.22} C_VEL
LIN {X 0,Y 608.478,Z 376.883,A -85,B 0,C 180,E1 -472.048,E2 -472.048} C_VEL
LIN {X 0,Y 608.492,Z 366.349,A -85,B 0,C 180,E1 -474.57,E2 -474.57} C_VEL
LIN {X 0,Y 608.515,Z 355.525,A -85,B 0,C 180,E1 -477.214,E2 -477.214} C_VEL
LIN {X 0,Y 608.521,Z 345.281,A -85,B 0,C 180,E1 -479.777,E2 -479.777} C_VEL
LIN {X 0,Y 608.555,Z 334.533,A -85,B 0,C 180,E1 -482.536,E2 -482.536} C_VEL
LIN {X 0,Y 608.59,Z 327.291,A -85,B 0,C 180,E1 -484.462,E2 -484.462} C_VEL
LIN {X 0,Y 608.443,Z 325.319,A -85,B 0,C 180,E1 -485.061,E2 -485.061} C_VEL
LIN {X 0,Y 608.474,Z 325.321,A -85,B 0,C 180,E1 -487.746,E2 -487.746} C_VEL
LIN {X 0,Y 608.451,Z 325.316,A -85,B 0,C 180,E1 -490.329,E2 -490.329} C_VEL
LIN {X 0,Y 608.484,Z 325.313,A -85,B 0,C 180,E1 -493.31,E2 -493.31} C_VEL
LIN {X 0,Y 608.468,Z 325.321,A -85,B 0,C 180,E1 -496.131,E2 -496.131} C_VEL
LIN {X 0,Y 608.451,Z 325.316,A -85,B 0,C 180,E1 -498.823,E2 -498.823} C_VEL
LIN {X 0,Y 608.472,Z 325.318,A -85,B 0,C 180,E1 -501.412,E2 -501.412} C_VEL
LIN {X 0,Y 608.481,Z 325.312,A -85,B 0,C 180,E1 -503.951,E2 -503.951} C_VEL
LIN {X 0,Y 608.45,Z 325.323,A -85,B 0,C 180,E1 -506.328,E2 -506.328} C_VEL
LIN {X 0,Y 608.449,Z 325.316,A -85,B 0,C 180,E1 -508.733,E2 -508.733} C_VEL
LIN {X 0,Y 608.477,Z 325.319,A -85,B 0,C 180,E1 -511.38,E2 -511.38} C_VEL
LIN {X 0,Y 608.443,Z 325.317,A -85,B 0,C 180,E1 -513.964,E2 -513.964} C_VEL
LIN {X 0,Y 608.475,Z 325.317,A -85,B 0,C 180,E1 -516.156,E2 -516.156} C_VEL
LIN {X 0,Y 608.451,Z 325.316,A -85,B 0,C 180,E1 -519.018,E2 -519.018} C_VEL
LIN {X 0,Y 608.448,Z 325.318,A -85,B 0,C 180,E1 -521.828,E2 -521.828} C_VEL
LIN {X 0,Y 608.472,Z 325.318,A -85,B 0,C 180,E1 -524.594,E2 -524.594} C_VEL
LIN {X 0,Y 608.476,Z 325.312,A -85,B 0,C 180,E1 -527.323,E2 -527.323} C_VEL
LIN {X 0,Y 608.453,Z 325.32,A -85,B 0,C 180,E1 -530.023,E2 -530.023} C_VEL
LIN {X 0,Y 608.468,Z 325.315,A -85,B 0,C 180,E1 -532.701,E2 -532.701} C_VEL
LIN {X 0,Y 608.459,Z 325.316,A -85,B 0,C 180,E1 -535.362,E2 -535.362} C_VEL
LIN {X 0,Y 608.462,Z 325.319,A -85,B 0,C 180,E1 -538.014,E2 -538.014} C_VEL
LIN {X 0,Y 608.478,Z 325.312,A -85,B 0,C 180,E1 -540.662,E2 -540.662} C_VEL
LIN {X 0,Y 608.482,Z 325.319,A -85,B 0,C 180,E1 -543.311,E2 -543.311} C_VEL
LIN {X 0,Y 608.454,Z 325.316,A -85,B 0,C 180,E1 -545.967,E2 -545.967} C_VEL
LIN {X 0,Y 608.455,Z 325.318,A -85,B 0,C 180,E1 -548.636,E2 -548.636} C_VEL
LIN {X 0,Y 608.463,Z 325.315,A -85,B 0,C 180,E1 -549.46,E2 -549.46} C_VEL
LIN {X 0,Y 607.785,Z 325.406,A -85,B 0,C 180,E1 -550.013,E2 -550.013} C_VEL
LIN {X 0,Y 604.932,Z 325.759,A -85,B 0,C 180,E1 -550.91,E2 -550.91} C_VEL
LIN {X 0,Y 602.529,Z 326.061,A -85,B 0,C 180,E1 -551.631,E2 -551.631} C_VEL
LIN {X 0,Y 601.497,Z 326.183,A -85,B 0,C 180,E1 -552.188,E2 -552.188} C_VEL
LIN {X 0,Y 601.412,Z 326.193,A -85,B 0,C 180,E1 -552.376,E2 -552.376} C_VEL
LIN {X 0,Y 601.431,Z 326.196,A -85,B 0,C 180,E1 -554.897,E2 -554.897} C_VEL
LIN {X 0,Y 601.439,Z 326.193,A -85,B 0,C 180,E1 -556.986,E2 -556.986} C_VEL
LIN {X 0,Y 601.409,Z 326.197,A -85,B 0,C 180,E1 -559.809,E2 -559.809} C_VEL
LIN {X 0,Y 601.417,Z 326.192,A -85,B 0,C 180,E1 -562.683,E2 -562.683} C_VEL
LIN {X 0,Y 601.404,Z 326.197,A -85,B 0,C 180,E1 -564.879,E2 -564.879} C_VEL
LIN {X 0,Y 601.421,Z 326.192,A -85,B 0,C 180,E1 -567.363,E2 -567.363} C_VEL
LIN {X 0,Y 601.434,Z 326.198,A -85,B 0,C 180,E1 -570.164,E2 -570.164} C_VEL
LIN {X 0,Y 601.418,Z 326.192,A -85,B 0,C 180,E1 -572.714,E2 -572.714} C_VEL
LIN {X 0,Y 601.401,Z 326.2,A -85,B 0,C 180,E1 -575.112,E2 -575.112} C_VEL
LIN {X 0,Y 601.437,Z 326.19,A -85,B 0,C 180,E1 -577.419,E2 -577.419} C_VEL
LIN {X 0,Y 601.408,Z 326.197,A -85,B 0,C 180,E1 -579.996,E2 -579.996} C_VEL
LIN {X 0,Y 601.412,Z 326.193,A -85,B 0,C 180,E1 -582.67,E2 -582.67} C_VEL
LIN {X 0,Y 601.43,Z 326.195,A -85,B 0,C 180,E1 -585.482,E2 -585.482} C_VEL
LIN {X 0,Y 601.426,Z 326.195,A -85,B 0,C 180,E1 -588.407,E2 -588.407} C_VEL
LIN {X 0,Y 601.414,Z 326.194,A -85,B 0,C 180,E1 -590.873,E2 -590.873} C_VEL
LIN {X 0,Y 601.436,Z 326.329,A -85,B 0,C 180,E1 -591.733,E2 -591.733} C_VEL
LIN {X 0,Y 601.45,Z 331.246,A -85,B 0,C 180,E1 -594.249,E2 -594.249} C_VEL
LIN {X 0,Y 601.441,Z 336.067,A -85,B 0,C 180,E1 -596.687,E2 -596.687} C_VEL
LIN {X 0,Y 601.406,Z 340.832,A -85,B 0,C 180,E1 -599.057,E2 -599.057} C_VEL
LIN {X 0,Y 601.405,Z 345.639,A -85,B 0,C 180,E1 -601.372,E2 -601.372} C_VEL
LIN {X 0,Y 601.404,Z 352.053,A -85,B 0,C 180,E1 -604.381,E2 -604.381} C_VEL
LIN {X 0,Y 601.372,Z 358.467,A -85,B 0,C 180,E1 -607.315,E2 -607.315} C_VEL
LIN {X 0,Y 601.361,Z 364.882,A -85,B 0,C 180,E1 -610.189,E2 -610.189} C_VEL
LIN {X 0,Y 601.361,Z 371.297,A -85,B 0,C 180,E1 -613.012,E2 -613.012} C_VEL
LIN {X 0,Y 601.332,Z 377.475,A -85,B 0,C 180,E1 -615.69,E2 -615.69} C_VEL
LIN {X 0,Y 601.719,Z 380.864,A -85,B 0,C 180,E1 -615.749,E2 -615.749} C_VEL
LIN {X 0,Y 601.686,Z 394.954,A -85,B 0,C 180,E1 -616.038,E2 -616.038} C_VEL
LIN {X 0,Y 601.647,Z 407.63,A -85,B 0,C 180,E1 -616.421,E2 -616.421} C_VEL
LIN {X 0,Y 601.618,Z 420.063,A -85,B 0,C 180,E1 -616.919,E2 -616.919} C_VEL
LIN {X 0,Y 601.567,Z 431.952,A -85,B 0,C 180,E1 -617.518,E2 -617.518} C_VEL
LIN {X 0,Y 601.534,Z 444.308,A -85,B 0,C 180,E1 -618.288,E2 -618.288} C_VEL
LIN {X 0,Y 601.496,Z 455.305,A -85,B 0,C 180,E1 -619.124,E2 -619.124} C_VEL
LIN {X 0,Y 601.435,Z 465.65,A -85,B 0,C 180,E1 -620.075,E2 -620.075} C_VEL
LIN {X 0,Y 601.411,Z 474.837,A -85,B 0,C 180,E1 -621.093,E2 -621.093} C_VEL
LIN {X 0,Y 601.387,Z 483.62,A -85,B 0,C 180,E1 -622.276,E2 -622.276} C_VEL
LIN {X 0,Y 601.373,Z 490.382,A -85,B 0,C 180,E1 -623.395,E2 -623.395} C_VEL
LIN {X 0,Y 601.354,Z 496.378,A -85,B 0,C 180,E1 -624.635,E2 -624.635} C_VEL
LIN {X 0,Y 601.345,Z 501.3,A -85,B 0,C 180,E1 -625.979,E2 -625.979} C_VEL
LIN {X 0,Y 601.324,Z 504.735,A -85,B 0,C 180,E1 -627.32,E2 -627.32} C_VEL
LIN {X 0,Y 601.346,Z 506.779,A -85,B 0,C 180,E1 -628.661,E2 -628.661} C_VEL
LIN {X 0,Y 601.334,Z 507.496,A -85,B 0,C 180,E1 -630,E2 -630} C_VEL
LIN {X 0,Y 601.343,Z 506.882,A -85,B 0,C 180,E1 -631.339,E2 -631.339} C_VEL
LIN {X 0,Y 601.321,Z 504.928,A -85,B 0,C 180,E1 -632.68,E2 -632.68} C_VEL
LIN {X 0,Y 601.346,Z 501.583,A -85,B 0,C 180,E1 -634.021,E2 -634.021} C_VEL
LIN {X 0,Y 601.355,Z 496.757,A -85,B 0,C 180,E1 -635.365,E2 -635.365} C_VEL
LIN {X 0,Y 601.368,Z 490.888,A -85,B 0,C 180,E1 -636.601,E2 -636.601} C_VEL
LIN {X 0,Y 601.386,Z 484.216,A -85,B 0,C 180,E1 -637.724,E2 -637.724} C_VEL
LIN {X 0,Y 601.411,Z 475.558,A -85,B 0,C 180,E1 -638.908,E2 -638.908} C_VEL
LIN {X 0,Y 601.432,Z 466.511,A -85,B 0,C 180,E1 -639.925,E2 -639.925} C_VEL
LIN {X 0,Y 601.474,Z 455.335,A -85,B 0,C 180,E1 -640.964,E2 -640.964} C_VEL
LIN {X 0,Y 601.547,Z 443.095,A -85,B 0,C 180,E1 -641.883,E2 -641.883} C_VEL
LIN {X 0,Y 601.551,Z 430.461,A -85,B 0,C 180,E1 -642.654,E2 -642.654} C_VEL
LIN {X 0,Y 601.616,Z 418.185,A -85,B 0,C 180,E1 -643.253,E2 -643.253} C_VEL
LIN {X 0,Y 601.678,Z 404.207,A -85,B 0,C 180,E1 -643.782,E2 -643.782} C_VEL
LIN {X 0,Y 601.706,Z 390.529,A -85,B 0,C 180,E1 -644.156,E2 -644.156} C_VEL
LIN {X 0,Y 601.589,Z 378.973,A -85,B 0,C 180,E1 -644.371,E2 -644.371} C_VEL
LIN {X 0,Y 601.347,Z 377.47,A -85,B 0,C 180,E1 -644.402,E2 -644.402} C_VEL
LIN {X 0,Y 601.357,Z 371.503,A -85,B 0,C 180,E1 -646.988,E2 -646.988} C_VEL
LIN {X 0,Y 601.363,Z 365.084,A -85,B 0,C 180,E1 -649.811,E2 -649.811} C_VEL
LIN {X 0,Y 601.373,Z 358.666,A -85,B 0,C 180,E1 -652.685,E2 -652.685} C_VEL
LIN {X 0,Y 601.404,Z 352.247,A -85,B 0,C 180,E1 -655.619,E2 -655.619} C_VEL
LIN {X 0,Y 601.409,Z 345.828,A -85,B 0,C 180,E1 -658.628,E2 -658.628} C_VEL
LIN {X 0,Y 601.424,Z 339.983,A -85,B 0,C 180,E1 -661.455,E2 -661.455} C_VEL
LIN {X 0,Y 601.433,Z 334.631,A -85,B 0,C 180,E1 -664.118,E2 -664.118} C_VEL
LIN {X 0,Y 601.44,Z 329.796,A -85,B 0,C 180,E1 -666.581,E2 -666.581} C_VEL
LIN {X 0,Y 601.439,Z 326.194,A -85,B 0,C 180,E1 -668.471,E2 -668.471} C_VEL
LIN {X 0,Y 601.428,Z 326.196,A -85,B 0,C 180,E1 -671.593,E2 -671.593} C_VEL
LIN {X 0,Y 601.43,Z 326.194,A -85,B 0,C 180,E1 -674.535,E2 -674.535} C_VEL
LIN {X 0,Y 601.413,Z 326.192,A -85,B 0,C 180,E1 -677.41,E2 -677.41} C_VEL
LIN {X 0,Y 601.408,Z 326.198,A -85,B 0,C 180,E1 -680.004,E2 -680.004} C_VEL
LIN {X 0,Y 601.439,Z 326.19,A -85,B 0,C 180,E1 -682.618,E2 -682.618} C_VEL
LIN {X 0,Y 601.434,Z 326.19,A -85,B 0,C 180,E1 -685.882,E2 -685.882} C_VEL
LIN {X 0,Y 601.425,Z 326.194,A -85,B 0,C 180,E1 -688.546,E2 -688.546} C_VEL
LIN {X 0,Y 601.441,Z 326.193,A -85,B 0,C 180,E1 -691.373,E2 -691.373} C_VEL
LIN {X 0,Y 601.403,Z 326.196,A -85,B 0,C 180,E1 -693.636,E2 -693.636} C_VEL
LIN {X 0,Y 601.421,Z 326.199,A -85,B 0,C 180,E1 -696.59,E2 -696.59} C_VEL
LIN {X 0,Y 601.429,Z 326.191,A -85,B 0,C 180,E1 -699.478,E2 -699.478} C_VEL
LIN {X 0,Y 601.398,Z 326.195,A -85,B 0,C 180,E1 -702.312,E2 -702.312} C_VEL
LIN {X 0,Y 601.417,Z 326.192,A -85,B 0,C 180,E1 -704.409,E2 -704.409} C_VEL
LIN {X 0,Y 601.422,Z 326.193,A -85,B 0,C 180,E1 -707.172,E2 -707.172} C_VEL
LIN {X 0,Y 601.44,Z 326.194,A -85,B 0,C 180,E1 -709.905,E2 -709.905} C_VEL
LIN {X 0,Y 601.444,Z 326.188,A -85,B 0,C 180,E1 -712.615,E2 -712.615} C_VEL
LIN {X 0,Y 601.431,Z 326.195,A -85,B 0,C 180,E1 -715.308,E2 -715.308} C_VEL
LIN {X 0,Y 601.42,Z 326.193,A -85,B 0,C 180,E1 -717.991,E2 -717.991} C_VEL
LIN {X 0,Y 601.451,Z 326.189,A -85,B 0,C 180,E1 -720.669,E2 -720.669} C_VEL
LIN {X 0,Y 601.43,Z 326.195,A -85,B 0,C 180,E1 -723.349,E2 -723.349} C_VEL
LIN {X 0,Y 601.409,Z 326.193,A -85,B 0,C 180,E1 -726.037,E2 -726.037} C_VEL
LIN {X 0,Y 601.42,Z 326.196,A -85,B 0,C 180,E1 -728.738,E2 -728.738} C_VEL
LIN {X 0,Y 601.44,Z 326.191,A -85,B 0,C 180,E1 -731.458,E2 -731.458} C_VEL
LIN {X 0,Y 601.426,Z 326.191,A -85,B 0,C 180,E1 -734.205,E2 -734.205} C_VEL
LIN {X 0,Y 601.437,Z 326.197,A -85,B 0,C 180,E1 -736.986,E2 -736.986} C_VEL
LIN {X 0,Y 601.408,Z 326.194,A -85,B 0,C 180,E1 -739.809,E2 -739.809} C_VEL
LIN {X 0,Y 601.418,Z 326.192,A -85,B 0,C 180,E1 -742.683,E2 -742.683} C_VEL
LIN {X 0,Y 601.407,Z 326.195,A -85,B 0,C 180,E1 -744.878,E2 -744.878} C_VEL
LIN {X 0,Y 601.421,Z 326.194,A -85,B 0,C 180,E1 -747.362,E2 -747.362} C_VEL
LIN {X 0,Y 601.433,Z 326.194,A -85,B 0,C 180,E1 -750.164,E2 -750.164} C_VEL
LIN {X 0,Y 601.417,Z 326.192,A -85,B 0,C 180,E1 -752.714,E2 -752.714} C_VEL
LIN {X 0,Y 601.417,Z 326.195,A -85,B 0,C 180,E1 -755.114,E2 -755.114} C_VEL
LIN {X 0,Y 601.44,Z 326.192,A -85,B 0,C 180,E1 -757.419,E2 -757.419} C_VEL
LIN {X 0,Y 601.407,Z 326.195,A -85,B 0,C 180,E1 -759.995,E2 -759.995} C_VEL
LIN {X 0,Y 601.41,Z 326.194,A -85,B 0,C 180,E1 -762.67,E2 -762.67} C_VEL
LIN {X 0,Y 601.43,Z 326.198,A -85,B 0,C 180,E1 -765.482,E2 -765.482} C_VEL
LIN {X 0,Y 601.427,Z 326.193,A -85,B 0,C 180,E1 -768.406,E2 -768.406} C_VEL
LIN {X 0,Y 601.435,Z 326.191,A -85,B 0,C 180,E1 -771.529,E2 -771.529} C_VEL
LIN {X 0,Y 601.388,Z 326.202,A -85,B 0,C 180,E1 -774.245,E2 -774.245} C_VEL
LIN {X 0,Y 601.408,Z 326.284,A -85,B 0,C 180,E1 -774.771,E2 -774.771} C_VEL
LIN {X 0,Y 601.668,Z 330.803,A -85,B 0,C 180,E1 -776.031,E2 -776.031} C_VEL
LIN {X 0,Y 601.614,Z 341.198,A -85,B 0,C 180,E1 -778.79,E2 -778.79} C_VEL
LIN {X 0,Y 601.569,Z 352.804,A -85,B 0,C 180,E1 -781.761,E2 -781.761} C_VEL
LIN {X 0,Y 601.507,Z 363.339,A -85,B 0,C 180,E1 -784.386,E2 -784.386} C_VEL
LIN {X 0,Y 601.503,Z 375.378,A -85,B 0,C 180,E1 -787.32,E2 -787.32} C_VEL
LIN {X 0,Y 601.444,Z 387.417,A -85,B 0,C 180,E1 -790.192,E2 -790.192} C_VEL
LIN {X 0,Y 601.423,Z 400.271,A -85,B 0,C 180,E1 -793.203,E2 -793.203} C_VEL
LIN {X 0,Y 601.908,Z 403.913,A -85,B 0,C 180,E1 -793.272,E2 -793.272} C_VEL
LIN {X 0,Y 601.862,Z 419.044,A -85,B 0,C 180,E1 -793.521,E2 -793.521} C_VEL
LIN {X 0,Y 601.824,Z 433.797,A -85,B 0,C 180,E1 -793.898,E2 -793.898} C_VEL
LIN {X 0,Y 601.734,Z 448.665,A -85,B 0,C 180,E1 -794.417,E2 -794.417} C_VEL
LIN {X 0,Y 601.72,Z 462.109,A -85,B 0,C 180,E1 -795.024,E2 -795.024} C_VEL
LIN {X 0,Y 601.64,Z 476.033,A -85,B 0,C 180,E1 -795.8,E2 -795.8} C_VEL
LIN {X 0,Y 601.561,Z 488.691,A -85,B 0,C 180,E1 -796.659,E2 -796.659} C_VEL
LIN {X 0,Y 601.522,Z 499.333,A -85,B 0,C 180,E1 -797.517,E2 -797.517} C_VEL
LIN {X 0,Y 601.457,Z 510.138,A -85,B 0,C 180,E1 -798.542,E2 -798.542} C_VEL
LIN {X 0,Y 601.429,Z 520.658,A -85,B 0,C 180,E1 -799.735,E2 -799.735} C_VEL
LIN {X 0,Y 601.391,Z 529.411,A -85,B 0,C 180,E1 -800.923,E2 -800.923} C_VEL
LIN {X 0,Y 601.403,Z 535.752,A -85,B 0,C 180,E1 -801.939,E2 -801.939} C_VEL
LIN {X 0,Y 601.366,Z 543.222,A -85,B 0,C 180,E1 -803.399,E2 -803.399} C_VEL
LIN {X 0,Y 601.353,Z 548.161,A -85,B 0,C 180,E1 -804.635,E2 -804.635} C_VEL
LIN {X 0,Y 601.338,Z 552.288,A -85,B 0,C 180,E1 -805.979,E2 -805.979} C_VEL
LIN {X 0,Y 601.323,Z 555.185,A -85,B 0,C 180,E1 -807.32,E2 -807.32} C_VEL
LIN {X 0,Y 601.345,Z 556.913,A -85,B 0,C 180,E1 -808.661,E2 -808.661} C_VEL
LIN {X 0,Y 601.332,Z 557.5,A -85,B 0,C 180,E1 -810,E2 -810} C_VEL
LIN {X 0,Y 601.345,Z 556.913,A -85,B 0,C 180,E1 -811.339,E2 -811.339} C_VEL
LIN {X 0,Y 601.323,Z 555.185,A -85,B 0,C 180,E1 -812.68,E2 -812.68} C_VEL
LIN {X 0,Y 601.338,Z 552.288,A -85,B 0,C 180,E1 -814.021,E2 -814.021} C_VEL
LIN {X 0,Y 601.353,Z 548.161,A -85,B 0,C 180,E1 -815.365,E2 -815.365} C_VEL
LIN {X 0,Y 601.353,Z 542.703,A -85,B 0,C 180,E1 -816.711,E2 -816.711} C_VEL
LIN {X 0,Y 601.403,Z 535.752,A -85,B 0,C 180,E1 -818.061,E2 -818.061} C_VEL
LIN {X 0,Y 601.394,Z 527.092,A -85,B 0,C 180,E1 -819.416,E2 -819.416} C_VEL
LIN {X 0,Y 601.439,Z 517.877,A -85,B 0,C 180,E1 -820.605,E2 -820.605} C_VEL
LIN {X 0,Y 601.494,Z 508.509,A -85,B 0,C 180,E1 -821.628,E2 -821.628} C_VEL
LIN {X 0,Y 601.531,Z 497.388,A -85,B 0,C 180,E1 -822.654,E2 -822.654} C_VEL
LIN {X 0,Y 601.605,Z 484.466,A -85,B 0,C 180,E1 -823.649,E2 -823.649} C_VEL
LIN {X 0,Y 601.664,Z 471.782,A -85,B 0,C 180,E1 -824.459,E2 -824.459} C_VEL
LIN {X 0,Y 601.717,Z 458.609,A -85,B 0,C 180,E1 -825.15,E2 -825.15} C_VEL
LIN {X 0,Y 601.762,Z 444.182,A -85,B 0,C 180,E1 -825.756,E2 -825.756} C_VEL
LIN {X 0,Y 601.826,Z 429.25,A -85,B 0,C 180,E1 -826.233,E2 -826.233} C_VEL
LIN {X 0,Y 601.875,Z 414.198,A -85,B 0,C 180,E1 -826.571,E2 -826.571} C_VEL
LIN {X 0,Y 601.704,Z 401.923,A -85,B 0,C 180,E1 -826.758,E2 -826.758} C_VEL
LIN {X 0,Y 601.412,Z 400.223,A -85,B 0,C 180,E1 -826.808,E2 -826.808} C_VEL
LIN {X 0,Y 601.444,Z 387.417,A -85,B 0,C 180,E1 -829.808,E2 -829.808} C_VEL
LIN {X 0,Y 601.502,Z 375.378,A -85,B 0,C 180,E1 -832.68,E2 -832.68} C_VEL
LIN {X 0,Y 601.507,Z 363.339,A -85,B 0,C 180,E1 -835.614,E2 -835.614} C_VEL
LIN {X 0,Y 601.569,Z 352.805,A -85,B 0,C 180,E1 -838.239,E2 -838.239} C_VEL
LIN {X 0,Y 601.614,Z 341.199,A -85,B 0,C 180,E1 -841.21,E2 -841.21} C_VEL
LIN {X 0,Y 601.669,Z 330.311,A -85,B 0,C 180,E1 -844.103,E2 -844.103} C_VEL
LIN {X 0,Y 601.413,Z 326.197,A -85,B 0,C 180,E1 -845.272,E2 -845.272} C_VEL
LIN {X 0,Y 601.425,Z 326.193,A -85,B 0,C 180,E1 -848.268,E2 -848.268} C_VEL
LIN {X 0,Y 601.418,Z 326.196,A -85,B 0,C 180,E1 -850.874,E2 -850.874} C_VEL
LIN {X 0,Y 601.452,Z 326.187,A -85,B 0,C 180,E1 -853.584,E2 -853.584} C_VEL
LIN {X 0,Y 601.431,Z 326.194,A -85,B 0,C 180,E1 -856.428,E2 -856.428} C_VEL
LIN {X 0,Y 601.416,Z 326.194,A -85,B 0,C 180,E1 -859.126,E2 -859.126} C_VEL
LIN {X 0,Y 601.422,Z 326.193,A -85,B 0,C 180,E1 -861.732,E2 -861.732} C_VEL
LIN {X 0,Y 601.412,Z 326.196,A -85,B 0,C 180,E1 -864.247,E2 -864.247} C_VEL
LIN {X 0,Y 601.418,Z 326.194,A -85,B 0,C 180,E1 -866.686,E2 -866.686} C_VEL
LIN {X 0,Y 601.418,Z 326.193,A -85,B 0,C 180,E1 -869.058,E2 -869.058} C_VEL
LIN {X 0,Y 601.436,Z 326.196,A -85,B 0,C 180,E1 -871.373,E2 -871.373} C_VEL
LIN {X 0,Y 601.404,Z 326.194,A -85,B 0,C 180,E1 -873.636,E2 -873.636} C_VEL
LIN {X 0,Y 601.424,Z 326.195,A -85,B 0,C 180,E1 -876.59,E2 -876.59} C_VEL
LIN {X 0,Y 601.428,Z 326.194,A -85,B 0,C 180,E1 -879.478,E2 -879.478} C_VEL
LIN {X 0,Y 601.399,Z 326.194,A -85,B 0,C 180,E1 -882.312,E2 -882.312} C_VEL
LIN {X 0,Y 601.414,Z 326.195,A -85,B 0,C 180,E1 -884.409,E2 -884.409} C_VEL
LIN {X 0,Y 601.422,Z 326.191,A -85,B 0,C 180,E1 -887.172,E2 -887.172} C_VEL
LIN {X 0,Y 601.431,Z 326.196,A -85,B 0,C 180,E1 -889.905,E2 -889.905} C_VEL
LIN {X 0,Y 601.445,Z 326.189,A -85,B 0,C 180,E1 -892.615,E2 -892.615} C_VEL
LIN {X 0,Y 601.428,Z 326.192,A -85,B 0,C 180,E1 -895.308,E2 -895.308} C_VEL
LIN {X 0,Y 601.431,Z 326.194,A -85,B 0,C 180,E1 -897.991,E2 -897.991} C_VEL
LIN {X 0,Y 601.45,Z 326.187,A -85,B 0,C 180,E1 -900.67,E2 -900.67} C_VEL
LIN {X 0,Y 601.432,Z 326.196,A -85,B 0,C 180,E1 -903.35,E2 -903.35} C_VEL
LIN {X 0,Y 601.409,Z 326.194,A -85,B 0,C 180,E1 -906.037,E2 -906.037} C_VEL
LIN {X 0,Y 601.417,Z 326.194,A -85,B 0,C 180,E1 -908.738,E2 -908.738} C_VEL
LIN {X 0,Y 601.439,Z 326.193,A -85,B 0,C 180,E1 -911.458,E2 -911.458} C_VEL
LIN {X 0,Y 601.412,Z 326.193,A -85,B 0,C 180,E1 -912.376,E2 -912.376} C_VEL
LIN {X 0,Y 600.746,Z 326.278,A -85,B 0,C 180,E1 -912.936,E2 -912.936} C_VEL
LIN {X 0,Y 597.895,Z 326.636,A -85,B 0,C 180,E1 -913.843,E2 -913.843} C_VEL
LIN {X 0,Y 595.486,Z 326.939,A -85,B 0,C 180,E1 -914.574,E2 -914.574} C_VEL
LIN {X 0,Y 594.449,Z 327.066,A -85,B 0,C 180,E1 -915.137,E2 -915.137} C_VEL
LIN {X 0,Y 594.363,Z 327.074,A -85,B 0,C 180,E1 -915.328,E2 -915.328} C_VEL
LIN {X 0,Y 594.395,Z 327.068,A -85,B 0,C 180,E1 -917.193,E2 -917.193} C_VEL
LIN {X 0,Y 594.377,Z 327.076,A -85,B 0,C 180,E1 -920.054,E2 -920.054} C_VEL
LIN {X 0,Y 594.368,Z 327.071,A -85,B 0,C 180,E1 -922.967,E2 -922.967} C_VEL
LIN {X 0,Y 594.375,Z 327.076,A -85,B 0,C 180,E1 -925.193,E2 -925.193} C_VEL
LIN {X 0,Y 594.391,Z 327.067,A -85,B 0,C 180,E1 -927.527,E2 -927.527} C_VEL
LIN {X 0,Y 594.391,Z 327.072,A -85,B 0,C 180,E1 -930.328,E2 -930.328} C_VEL
LIN {X 0,Y 594.382,Z 327.069,A -85,B 0,C 180,E1 -932.95,E2 -932.95} C_VEL
LIN {X 0,Y 594.355,Z 327.076,A -85,B 0,C 180,E1 -935.409,E2 -935.409} C_VEL
LIN {X 0,Y 594.388,Z 327.068,A -85,B 0,C 180,E1 -937.941,E2 -937.941} C_VEL
LIN {X 0,Y 594.38,Z 327.069,A -85,B 0,C 180,E1 -940.822,E2 -940.822} C_VEL
LIN {X 0,Y 594.371,Z 327.074,A -85,B 0,C 180,E1 -943.839,E2 -943.839} C_VEL
LIN {X 0,Y 594.372,Z 327.074,A -85,B 0,C 180,E1 -946.701,E2 -946.701} C_VEL
LIN {X 0,Y 594.37,Z 327.07,A -85,B 0,C 180,E1 -949.433,E2 -949.433} C_VEL
LIN {X 0,Y 594.409,Z 327.274,A -85,B 0,C 180,E1 -951.68,E2 -951.68} C_VEL
LIN {X 0,Y 594.429,Z 333.037,A -85,B 0,C 180,E1 -954.666,E2 -954.666} C_VEL
LIN {X 0,Y 594.385,Z 337.784,A -85,B 0,C 180,E1 -957.088,E2 -957.088} C_VEL
LIN {X 0,Y 594.372,Z 342.944,A -85,B 0,C 180,E1 -959.675,E2 -959.675} C_VEL
LIN {X 0,Y 594.335,Z 348.847,A -85,B 0,C 180,E1 -962.537,E2 -962.537} C_VEL
LIN {X 0,Y 594.323,Z 353.658,A -85,B 0,C 180,E1 -964.804,E2 -964.804} C_VEL
LIN {X 0,Y 594.29,Z 360.072,A -85,B 0,C 180,E1 -967.764,E2 -967.764} C_VEL
LIN {X 0,Y 594.268,Z 364.883,A -85,B 0,C 180,E1 -969.942,E2 -969.942} C_VEL
LIN {X 0,Y 594.27,Z 369.694,A -85,B 0,C 180,E1 -972.092,E2 -972.092} C_VEL
LIN {X 0,Y 594.255,Z 374.506,A -85,B 0,C 180,E1 -974.216,E2 -974.216} C_VEL
LIN {X 0,Y 594.3,Z 377.606,A -85,B 0,C 180,E1 -975.52,E2 -975.52} C_VEL
LIN {X 0,Y 594.85,Z 382.446,A -85,B 0,C 180,E1 -975.605,E2 -975.605} C_VEL
LIN {X 0,Y 594.801,Z 396.723,A -85,B 0,C 180,E1 -975.921,E2 -975.921} C_VEL
LIN {X 0,Y 594.742,Z 410.673,A -85,B 0,C 180,E1 -976.373,E2 -976.373} C_VEL
LIN {X 0,Y 594.655,Z 423.728,A -85,B 0,C 180,E1 -976.936,E2 -976.936} C_VEL
LIN {X 0,Y 594.59,Z 436.362,A -85,B 0,C 180,E1 -977.629,E2 -977.629} C_VEL
LIN {X 0,Y 594.515,Z 447.869,A -85,B 0,C 180,E1 -978.407,E2 -978.407} C_VEL
LIN {X 0,Y 594.474,Z 458.426,A -85,B 0,C 180,E1 -979.269,E2 -979.269} C_VEL
LIN {X 0,Y 594.392,Z 468.908,A -85,B 0,C 180,E1 -980.3,E2 -980.3} C_VEL
LIN {X 0,Y 594.355,Z 477.558,A -85,B 0,C 180,E1 -981.329,E2 -981.329} C_VEL
LIN {X 0,Y 594.314,Z 485.845,A -85,B 0,C 180,E1 -982.526,E2 -982.526} C_VEL
LIN {X 0,Y 594.271,Z 492.001,A -85,B 0,C 180,E1 -983.62,E2 -983.62} C_VEL
LIN {X 0,Y 594.245,Z 497.793,A -85,B 0,C 180,E1 -984.911,E2 -984.911} C_VEL
LIN {X 0,Y 594.261,Z 501.302,A -85,B 0,C 180,E1 -985.931,E2 -985.931} C_VEL
LIN {X 0,Y 594.224,Z 504.737,A -85,B 0,C 180,E1 -987.288,E2 -987.288} C_VEL
LIN {X 0,Y 594.245,Z 506.78,A -85,B 0,C 180,E1 -988.645,E2 -988.645} C_VEL
LIN {X 0,Y 594.235,Z 507.496,A -85,B 0,C 180,E1 -990,E2 -990} C_VEL
LIN {X 0,Y 594.242,Z 506.882,A -85,B 0,C 180,E1 -991.355,E2 -991.355} C_VEL
LIN {X 0,Y 594.222,Z 504.927,A -85,B 0,C 180,E1 -992.712,E2 -992.712} C_VEL
LIN {X 0,Y 594.262,Z 501.582,A -85,B 0,C 180,E1 -994.069,E2 -994.069} C_VEL
LIN {X 0,Y 594.275,Z 496.755,A -85,B 0,C 180,E1 -995.429,E2 -995.429} C_VEL
LIN {X 0,Y 594.277,Z 491.38,A -85,B 0,C 180,E1 -996.587,E2 -996.587} C_VEL
LIN {X 0,Y 594.316,Z 484.213,A -85,B 0,C 180,E1 -997.816,E2 -997.816} C_VEL
LIN {X 0,Y 594.368,Z 475.554,A -85,B 0,C 180,E1 -999.014,E2 -999.014} C_VEL
LIN {X 0,Y 594.4,Z 466.505,A -85,B 0,C 180,E1 -1000.044,E2 -1000.044} C_VEL
LIN {X 0,Y 594.478,Z 456.218,A -85,B 0,C 180,E1 -1001.017,E2 -1001.017} C_VEL
LIN {X 0,Y 594.549,Z 445.582,A -85,B 0,C 180,E1 -1001.852,E2 -1001.852} C_VEL
LIN {X 0,Y 594.605,Z 433.569,A -85,B 0,C 180,E1 -1002.631,E2 -1002.631} C_VEL
LIN {X 0,Y 594.681,Z 420.144,A -85,B 0,C 180,E1 -1003.324,E2 -1003.324} C_VEL
LIN {X 0,Y 594.774,Z 406.532,A -85,B 0,C 180,E1 -1003.866,E2 -1003.866} C_VEL
LIN {X 0,Y 594.802,Z 392.597,A -85,B 0,C 180,E1 -1004.273,E2 -1004.273} C_VEL
LIN {X 0,Y 594.635,Z 379.525,A -85,B 0,C 180,E1 -1004.534,E2 -1004.534} C_VEL
LIN {X 0,Y 594.289,Z 377.552,A -85,B 0,C 180,E1 -1004.571,E2 -1004.571} C_VEL
LIN {X 0,Y 594.29,Z 371.501,A -85,B 0,C 180,E1 -1007.197,E2 -1007.197} C_VEL
LIN {X 0,Y 594.286,Z 366.688,A -85,B 0,C 180,E1 -1009.337,E2 -1009.337} C_VEL
LIN {X 0,Y 594.286,Z 361.874,A -85,B 0,C 180,E1 -1011.507,E2 -1011.507} C_VEL
LIN {X 0,Y 594.333,Z 355.514,A -85,B 0,C 180,E1 -1014.421,E2 -1014.421} C_VEL
LIN {X 0,Y 594.302,Z 350.641,A -85,B 0,C 180,E1 -1016.704,E2 -1016.704} C_VEL
LIN {X 0,Y 594.345,Z 345.826,A -85,B 0,C 180,E1 -1019.001,E2 -1019.001} C_VEL
LIN {X 0,Y 594.382,Z 340.472,A -85,B 0,C 180,E1 -1021.643,E2 -1021.643} C_VEL
LIN {X 0,Y 594.402,Z 334.685,A -85,B 0,C 180,E1 -1024.579,E2 -1024.579} C_VEL
LIN {X 0,Y 594.418,Z 329.835,A -85,B 0,C 180,E1 -1027.085,E2 -1027.085} C_VEL
LIN {X 0,Y 594.392,Z 327.072,A -85,B 0,C 180,E1 -1028.58,E2 -1028.58} C_VEL
LIN {X 0,Y 594.385,Z 327.076,A -85,B 0,C 180,E1 -1031.464,E2 -1031.464} C_VEL
LIN {X 0,Y 594.383,Z 327.069,A -85,B 0,C 180,E1 -1034.237,E2 -1034.237} C_VEL
LIN {X 0,Y 594.364,Z 327.071,A -85,B 0,C 180,E1 -1037.149,E2 -1037.149} C_VEL
LIN {X 0,Y 594.376,Z 327.071,A -85,B 0,C 180,E1 -1039.433,E2 -1039.433} C_VEL
LIN {X 0,Y 594.394,Z 327.067,A -85,B 0,C 180,E1 -1042.392,E2 -1042.392} C_VEL
LIN {X 0,Y 594.386,Z 327.069,A -85,B 0,C 180,E1 -1045.42,E2 -1045.42} C_VEL
LIN {X 0,Y 594.381,Z 327.074,A -85,B 0,C 180,E1 -1048.358,E2 -1048.358} C_VEL
LIN {X 0,Y 594.39,Z 327.068,A -85,B 0,C 180,E1 -1051.042,E2 -1051.042} C_VEL
LIN {X 0,Y 594.388,Z 327.075,A -85,B 0,C 180,E1 -1053.3,E2 -1053.3} C_VEL
LIN {X 0,Y 594.393,Z 327.07,A -85,B 0,C 180,E1 -1056.296,E2 -1056.296} C_VEL
LIN {X 0,Y 594.403,Z 327.065,A -85,B 0,C 180,E1 -1059.224,E2 -1059.224} C_VEL
LIN {X 0,Y 594.355,Z 327.073,A -85,B 0,C 180,E1 -1062.095,E2 -1062.095} C_VEL
LIN {X 0,Y 594.371,Z 327.07,A -85,B 0,C 180,E1 -1064.219,E2 -1064.219} C_VEL
LIN {X 0,Y 594.369,Z 327.073,A -85,B 0,C 180,E1 -1067.017,E2 -1067.017} C_VEL
LIN {X 0,Y 594.398,Z 327.07,A -85,B 0,C 180,E1 -1069.784,E2 -1069.784} C_VEL
LIN {X 0,Y 594.398,Z 327.066,A -85,B 0,C 180,E1 -1072.527,E2 -1072.527} C_VEL
LIN {X 0,Y 594.4,Z 327.071,A -85,B 0,C 180,E1 -1075.252,E2 -1075.252} C_VEL
LIN {X 0,Y 594.391,Z 327.068,A -85,B 0,C 180,E1 -1077.967,E2 -1077.967} C_VEL
LIN {X 0,Y 594.423,Z 327.064,A -85,B 0,C 180,E1 -1080.677,E2 -1080.677} C_VEL
LIN {X 0,Y 594.381,Z 327.074,A -85,B 0,C 180,E1 -1083.389,E2 -1083.389} C_VEL
LIN {X 0,Y 594.366,Z 327.07,A -85,B 0,C 180,E1 -1086.109,E2 -1086.109} C_VEL
LIN {X 0,Y 594.387,Z 327.071,A -85,B 0,C 180,E1 -1088.842,E2 -1088.842} C_VEL
LIN {X 0,Y 594.399,Z 327.069,A -85,B 0,C 180,E1 -1091.595,E2 -1091.595} C_VEL
LIN {X 0,Y 594.395,Z 327.067,A -85,B 0,C 180,E1 -1094.377,E2 -1094.377} C_VEL
LIN {X 0,Y 594.394,Z 327.071,A -85,B 0,C 180,E1 -1097.193,E2 -1097.193} C_VEL
LIN {X 0,Y 594.376,Z 327.073,A -85,B 0,C 180,E1 -1100.054,E2 -1100.054} C_VEL
LIN {X 0,Y 594.37,Z 327.07,A -85,B 0,C 180,E1 -1102.967,E2 -1102.967} C_VEL
LIN {X 0,Y 594.381,Z 327.074,A -85,B 0,C 180,E1 -1105.193,E2 -1105.193} C_VEL
LIN {X 0,Y 594.391,Z 327.068,A -85,B 0,C 180,E1 -1107.526,E2 -1107.526} C_VEL
LIN {X 0,Y 594.391,Z 327.074,A -85,B 0,C 180,E1 -1110.328,E2 -1110.328} C_VEL
LIN {X 0,Y 594.38,Z 327.069,A -85,B 0,C 180,E1 -1112.95,E2 -1112.95} C_VEL
LIN {X 0,Y 594.385,Z 327.076,A -85,B 0,C 180,E1 -1115.407,E2 -1115.407} C_VEL
LIN {X 0,Y 594.389,Z 327.068,A -85,B 0,C 180,E1 -1117.94,E2 -1117.94} C_VEL
LIN {X 0,Y 594.38,Z 327.071,A -85,B 0,C 180,E1 -1120.822,E2 -1120.822} C_VEL
LIN {X 0,Y 594.368,Z 327.072,A -85,B 0,C 180,E1 -1123.299,E2 -1123.299} C_VEL
LIN {X 0,Y 594.386,Z 327.069,A -85,B 0,C 180,E1 -1126.159,E2 -1126.159} C_VEL
LIN {X 0,Y 594.382,Z 327.072,A -85,B 0,C 180,E1 -1129.177,E2 -1129.177} C_VEL
LIN {X 0,Y 594.39,Z 327.073,A -85,B 0,C 180,E1 -1132.059,E2 -1132.059} C_VEL
LIN {X 0,Y 594.399,Z 327.247,A -85,B 0,C 180,E1 -1134.542,E2 -1134.542} C_VEL
LIN {X 0,Y 594.792,Z 330.34,A -85,B 0,C 180,E1 -1135.447,E2 -1135.447} C_VEL
LIN {X 0,Y 594.706,Z 340.916,A -85,B 0,C 180,E1 -1138.306,E2 -1138.306} C_VEL
LIN {X 0,Y 594.598,Z 351.299,A -85,B 0,C 180,E1 -1141.013,E2 -1141.013} C_VEL
LIN {X 0,Y 594.553,Z 361.769,A -85,B 0,C 180,E1 -1143.67,E2 -1143.67} C_VEL
LIN {X 0,Y 594.505,Z 373.873,A -85,B 0,C 180,E1 -1146.67,E2 -1146.67} C_VEL
LIN {X 0,Y 594.433,Z 384.407,A -85,B 0,C 180,E1 -1149.225,E2 -1149.225} C_VEL
LIN {X 0,Y 594.375,Z 396.446,A -85,B 0,C 180,E1 -1152.095,E2 -1152.095} C_VEL
LIN {X 0,Y 594.378,Z 400.316,A -85,B 0,C 180,E1 -1153.009,E2 -1153.009} C_VEL
LIN {X 0,Y 595.125,Z 404.303,A -85,B 0,C 180,E1 -1153.081,E2 -1153.081} C_VEL
LIN {X 0,Y 595.066,Z 420.051,A -85,B 0,C 180,E1 -1153.348,E2 -1153.348} C_VEL
LIN {X 0,Y 594.991,Z 435.29,A -85,B 0,C 180,E1 -1153.752,E2 -1153.752} C_VEL
LIN {X 0,Y 594.867,Z 449.788,A -85,B 0,C 180,E1 -1154.276,E2 -1154.276} C_VEL
LIN {X 0,Y 594.796,Z 463.86,A -85,B 0,C 180,E1 -1154.933,E2 -1154.933} C_VEL
LIN {X 0,Y 594.691,Z 477.355,A -85,B 0,C 180,E1 -1155.712,E2 -1155.712} C_VEL
LIN {X 0,Y 594.587,Z 489.853,A -85,B 0,C 180,E1 -1156.587,E2 -1156.587} C_VEL
LIN {X 0,Y 594.535,Z 501.273,A -85,B 0,C 180,E1 -1157.541,E2 -1157.541} C_VEL
LIN {X 0,Y 594.434,Z 511.708,A -85,B 0,C 180,E1 -1158.572,E2 -1158.572} C_VEL
LIN {X 0,Y 594.38,Z 522.019,A -85,B 0,C 180,E1 -1159.784,E2 -1159.784} C_VEL
LIN {X 0,Y 594.338,Z 530.533,A -85,B 0,C 180,E1 -1160.986,E2 -1160.986} C_VEL
LIN {X 0,Y 594.31,Z 537.611,A -85,B 0,C 180,E1 -1162.184,E2 -1162.184} C_VEL
LIN {X 0,Y 594.262,Z 544.491,A -85,B 0,C 180,E1 -1163.623,E2 -1163.623} C_VEL
LIN {X 0,Y 594.245,Z 549.324,A -85,B 0,C 180,E1 -1164.911,E2 -1164.911} C_VEL
LIN {X 0,Y 594.251,Z 552.288,A -85,B 0,C 180,E1 -1165.931,E2 -1165.931} C_VEL
LIN {X 0,Y 594.223,Z 555.186,A -85,B 0,C 180,E1 -1167.288,E2 -1167.288} C_VEL
LIN {X 0,Y 594.245,Z 556.913,A -85,B 0,C 180,E1 -1168.645,E2 -1168.645} C_VEL
LIN {X 0,Y 594.233,Z 557.5,A -85,B 0,C 180,E1 -1170,E2 -1170} C_VEL
LIN {X 0,Y 594.245,Z 556.912,A -85,B 0,C 180,E1 -1171.355,E2 -1171.355} C_VEL
LIN {X 0,Y 594.223,Z 555.185,A -85,B 0,C 180,E1 -1172.712,E2 -1172.712} C_VEL
LIN {X 0,Y 594.251,Z 552.288,A -85,B 0,C 180,E1 -1174.069,E2 -1174.069} C_VEL
LIN {X 0,Y 594.274,Z 548.162,A -85,B 0,C 180,E1 -1175.429,E2 -1175.429} C_VEL
LIN {X 0,Y 594.275,Z 542.703,A -85,B 0,C 180,E1 -1176.792,E2 -1176.792} C_VEL
LIN {X 0,Y 594.323,Z 535.751,A -85,B 0,C 180,E1 -1178.158,E2 -1178.158} C_VEL
LIN {X 0,Y 594.341,Z 527.091,A -85,B 0,C 180,E1 -1179.529,E2 -1179.529} C_VEL
LIN {X 0,Y 594.402,Z 517.877,A -85,B 0,C 180,E1 -1180.732,E2 -1180.732} C_VEL
LIN {X 0,Y 594.467,Z 508.509,A -85,B 0,C 180,E1 -1181.767,E2 -1181.767} C_VEL
LIN {X 0,Y 594.552,Z 497.387,A -85,B 0,C 180,E1 -1182.805,E2 -1182.805} C_VEL
LIN {X 0,Y 594.652,Z 484.646,A -85,B 0,C 180,E1 -1183.799,E2 -1183.799} C_VEL
LIN {X 0,Y 594.748,Z 471.781,A -85,B 0,C 180,E1 -1184.63,E2 -1184.63} C_VEL
LIN {X 0,Y 594.846,Z 458.607,A -85,B 0,C 180,E1 -1185.329,E2 -1185.329} C_VEL
LIN {X 0,Y 594.919,Z 444.181,A -85,B 0,C 180,E1 -1185.942,E2 -1185.942} C_VEL
LIN {X 0,Y 595.011,Z 429.25,A -85,B 0,C 180,E1 -1186.424,E2 -1186.424} C_VEL
LIN {X 0,Y 595.064,Z 413.903,A -85,B 0,C 180,E1 -1186.772,E2 -1186.772} C_VEL
LIN {X 0,Y 594.923,Z 403.025,A -85,B 0,C 180,E1 -1186.941,E2 -1186.941} C_VEL
LIN {X 0,Y 594.397,Z 400.226,A -85,B 0,C 180,E1 -1187.012,E2 -1187.012} C_VEL
LIN {X 0,Y 594.428,Z 387.417,A -85,B 0,C 180,E1 -1190.052,E2 -1190.052} C_VEL
LIN {X 0,Y 594.5,Z 375.378,A -85,B 0,C 180,E1 -1192.962,E2 -1192.962} C_VEL
LIN {X 0,Y 594.532,Z 362.881,A -85,B 0,C 180,E1 -1196.052,E2 -1196.052} C_VEL
LIN {X 0,Y 594.608,Z 352.805,A -85,B 0,C 180,E1 -1198.6,E2 -1198.6} C_VEL
LIN {X 0,Y 594.68,Z 342.277,A -85,B 0,C 180,E1 -1201.332,E2 -1201.332} C_VEL
LIN {X 0,Y 594.762,Z 331.667,A -85,B 0,C 180,E1 -1204.193,E2 -1204.193} C_VEL
LIN {X 0,Y 594.467,Z 327.656,A -85,B 0,C 180,E1 -1205.339,E2 -1205.339} C_VEL
LIN {X 0,Y 594.354,Z 327.078,A -85,B 0,C 180,E1 -1205.513,E2 -1205.513} C_VEL
LIN {X 0,Y 594.389,Z 327.074,A -85,B 0,C 180,E1 -1207.941,E2 -1207.941} C_VEL
LIN {X 0,Y 594.38,Z 327.072,A -85,B 0,C 180,E1 -1210.822,E2 -1210.822} C_VEL
LIN {X 0,Y 594.385,Z 327.068,A -85,B 0,C 180,E1 -1213.841,E2 -1213.841} C_VEL
LIN {X 0,Y 594.368,Z 327.072,A -85,B 0,C 180,E1 -1216.701,E2 -1216.701} C_VEL
LIN {X 0,Y 594.375,Z 327.074,A -85,B 0,C 180,E1 -1219.434,E2 -1219.434} C_VEL
LIN {X 0,Y 594.393,Z 327.068,A -85,B 0,C 180,E1 -1222.392,E2 -1222.392} C_VEL
LIN {X 0,Y 594.388,Z 327.074,A -85,B 0,C 180,E1 -1224.672,E2 -1224.672} C_VEL
LIN {X 0,Y 594.379,Z 327.069,A -85,B 0,C 180,E1 -1227.089,E2 -1227.089} C_VEL
LIN {X 0,Y 594.39,Z 327.075,A -85,B 0,C 180,E1 -1229.672,E2 -1229.672} C_VEL
LIN {X 0,Y 594.379,Z 327.07,A -85,B 0,C 180,E1 -1232.539,E2 -1232.539} C_VEL
LIN {X 0,Y 594.38,Z 327.074,A -85,B 0,C 180,E1 -1234.807,E2 -1234.807} C_VEL
LIN {X 0,Y 594.369,Z 327.07,A -85,B 0,C 180,E1 -1237.265,E2 -1237.265} C_VEL
LIN {X 0,Y 594.376,Z 327.073,A -85,B 0,C 180,E1 -1239.946,E2 -1239.946} C_VEL
LIN {X 0,Y 594.393,Z 327.07,A -85,B 0,C 180,E1 -1242.807,E2 -1242.807} C_VEL
LIN {X 0,Y 594.394,Z 327.067,A -85,B 0,C 180,E1 -1245.827,E2 -1245.827} C_VEL
LIN {X 0,Y 594.399,Z 327.07,A -85,B 0,C 180,E1 -1248.405,E2 -1248.405} C_VEL
LIN {X 0,Y 594.385,Z 327.071,A -85,B 0,C 180,E1 -1251.158,E2 -1251.158} C_VEL
LIN {X 0,Y 594.366,Z 327.07,A -85,B 0,C 180,E1 -1253.891,E2 -1253.891} C_VEL
LIN {X 0,Y 594.381,Z 327.075,A -85,B 0,C 180,E1 -1256.611,E2 -1256.611} C_VEL
LIN {X 0,Y 594.422,Z 327.064,A -85,B 0,C 180,E1 -1259.323,E2 -1259.323} C_VEL
LIN {X 0,Y 594.392,Z 327.069,A -85,B 0,C 180,E1 -1262.033,E2 -1262.033} C_VEL
LIN {X 0,Y 594.401,Z 327.07,A -85,B 0,C 180,E1 -1264.748,E2 -1264.748} C_VEL
LIN {X 0,Y 594.397,Z 327.066,A -85,B 0,C 180,E1 -1267.473,E2 -1267.473} C_VEL
LIN {X 0,Y 594.397,Z 327.07,A -85,B 0,C 180,E1 -1270.216,E2 -1270.216} C_VEL
LIN {X 0,Y 594.369,Z 327.072,A -85,B 0,C 180,E1 -1272.983,E2 -1272.983} C_VEL
LIN {X 0,Y 594.363,Z 327.074,A -85,B 0,C 180,E1 -1275.328,E2 -1275.328} C_VEL
LIN {X 0,Y 593.69,Z 327.155,A -85,B 0,C 180,E1 -1275.894,E2 -1275.894} C_VEL
LIN {X 0,Y 590.823,Z 327.517,A -85,B 0,C 180,E1 -1276.812,E2 -1276.812} C_VEL
LIN {X 0,Y 588.413,Z 327.818,A -85,B 0,C 180,E1 -1277.55,E2 -1277.55} C_VEL
LIN {X 0,Y 587.39,Z 327.943,A -85,B 0,C 180,E1 -1278.121,E2 -1278.121} C_VEL
LIN {X 0,Y 587.314,Z 327.951,A -85,B 0,C 180,E1 -1278.314,E2 -1278.314} C_VEL
LIN {X 0,Y 587.336,Z 327.946,A -85,B 0,C 180,E1 -1281.038,E2 -1281.038} C_VEL
LIN {X 0,Y 587.326,Z 327.952,A -85,B 0,C 180,E1 -1283.259,E2 -1283.259} C_VEL
LIN {X 0,Y 587.333,Z 327.948,A -85,B 0,C 180,E1 -1285.517,E2 -1285.517} C_VEL
LIN {X 0,Y 587.353,Z 327.944,A -85,B 0,C 180,E1 -1287.818,E2 -1287.818} C_VEL
LIN {X 0,Y 587.342,Z 327.948,A -85,B 0,C 180,E1 -1290.51,E2 -1290.51} C_VEL
LIN {X 0,Y 587.34,Z 327.951,A -85,B 0,C 180,E1 -1293.396,E2 -1293.396} C_VEL
LIN {X 0,Y 587.296,Z 327.951,A -85,B 0,C 180,E1 -1295.9,E2 -1295.9} C_VEL
LIN {X 0,Y 587.333,Z 327.953,A -85,B 0,C 180,E1 -1298.479,E2 -1298.479} C_VEL
LIN {X 0,Y 587.339,Z 327.946,A -85,B 0,C 180,E1 -1301.157,E2 -1301.157} C_VEL
LIN {X 0,Y 587.331,Z 327.948,A -85,B 0,C 180,E1 -1304.113,E2 -1304.113} C_VEL
LIN {X 0,Y 587.32,Z 327.956,A -85,B 0,C 180,E1 -1306.994,E2 -1306.994} C_VEL
LIN {X 0,Y 587.315,Z 327.95,A -85,B 0,C 180,E1 -1309.745,E2 -1309.745} C_VEL
LIN {X 0,Y 587.346,Z 328.018,A -85,B 0,C 180,E1 -1311.522,E2 -1311.522} C_VEL
LIN {X 0,Y 587.381,Z 332.969,A -85,B 0,C 180,E1 -1314.106,E2 -1314.106} C_VEL
LIN {X 0,Y 587.346,Z 338.31,A -85,B 0,C 180,E1 -1316.888,E2 -1316.888} C_VEL
LIN {X 0,Y 587.323,Z 343.461,A -85,B 0,C 180,E1 -1319.493,E2 -1319.493} C_VEL
LIN {X 0,Y 587.276,Z 349.145,A -85,B 0,C 180,E1 -1322.322,E2 -1322.322} C_VEL
LIN {X 0,Y 587.25,Z 355.263,A -85,B 0,C 180,E1 -1325.237,E2 -1325.237} C_VEL
LIN {X 0,Y 587.248,Z 360.073,A -85,B 0,C 180,E1 -1327.482,E2 -1327.482} C_VEL
LIN {X 0,Y 587.195,Z 364.884,A -85,B 0,C 180,E1 -1329.69,E2 -1329.69} C_VEL
LIN {X 0,Y 587.182,Z 369.696,A -85,B 0,C 180,E1 -1331.869,E2 -1331.869} C_VEL
LIN {X 0,Y 587.175,Z 374.507,A -85,B 0,C 180,E1 -1334.021,E2 -1334.021} C_VEL
LIN {X 0,Y 587.217,Z 377.464,A -85,B 0,C 180,E1 -1335.333,E2 -1335.333} C_VEL
LIN {X 0,Y 587.984,Z 382.843,A -85,B 0,C 180,E1 -1335.441,E2 -1335.441} C_VEL
LIN {X 0,Y 587.917,Z 396.968,A -85,B 0,C 180,E1 -1335.759,E2 -1335.759} C_VEL
LIN {X 0,Y 587.825,Z 410.687,A -85,B 0,C 180,E1 -1336.209,E2 -1336.209} C_VEL
LIN {X 0,Y 587.726,Z 423.74,A -85,B 0,C 180,E1 -1336.78,E2 -1336.78} C_VEL
LIN {X 0,Y 587.622,Z 436.373,A -85,B 0,C 180,E1 -1337.48,E2 -1337.48} C_VEL
LIN {X 0,Y 587.514,Z 447.878,A -85,B 0,C 180,E1 -1338.267,E2 -1338.267} C_VEL
LIN {X 0,Y 587.467,Z 458.432,A -85,B 0,C 180,E1 -1339.139,E2 -1339.139} C_VEL
LIN {X 0,Y 587.355,Z 468.913,A -85,B 0,C 180,E1 -1340.183,E2 -1340.183} C_VEL
LIN {X 0,Y 587.311,Z 477.562,A -85,B 0,C 180,E1 -1341.224,E2 -1341.224} C_VEL
LIN {X 0,Y 587.25,Z 485.848,A -85,B 0,C 180,E1 -1342.435,E2 -1342.435} C_VEL
LIN {X 0,Y 587.181,Z 492.471,A -85,B 0,C 180,E1 -1343.636,E2 -1343.636} C_VEL
LIN {X 0,Y 587.158,Z 497.795,A -85,B 0,C 180,E1 -1344.85,E2 -1344.85} C_VEL
LIN {X 0,Y 587.181,Z 501.304,A -85,B 0,C 180,E1 -1345.882,E2 -1345.882} C_VEL
LIN {X 0,Y 587.13,Z 504.738,A -85,B 0,C 180,E1 -1347.256,E2 -1347.256} C_VEL
LIN {X 0,Y 587.145,Z 506.781,A -85,B 0,C 180,E1 -1348.628,E2 -1348.628} C_VEL
LIN {X 0,Y 587.136,Z 507.496,A -85,B 0,C 180,E1 -1350,E2 -1350} C_VEL
LIN {X 0,Y 587.142,Z 506.882,A -85,B 0,C 180,E1 -1351.372,E2 -1351.372} C_VEL
LIN {X 0,Y 587.128,Z 504.927,A -85,B 0,C 180,E1 -1352.744,E2 -1352.744} C_VEL
LIN {X 0,Y 587.182,Z 501.581,A -85,B 0,C 180,E1 -1354.118,E2 -1354.118} C_VEL
LIN {X 0,Y 587.2,Z 496.752,A -85,B 0,C 180,E1 -1355.495,E2 -1355.495} C_VEL
LIN {X 0,Y 587.21,Z 490.288,A -85,B 0,C 180,E1 -1356.874,E2 -1356.874} C_VEL
LIN {X 0,Y 587.269,Z 483.089,A -85,B 0,C 180,E1 -1358.084,E2 -1358.084} C_VEL
LIN {X 0,Y 587.332,Z 475.55,A -85,B 0,C 180,E1 -1359.123,E2 -1359.123} C_VEL
LIN {X 0,Y 587.376,Z 466.5,A -85,B 0,C 180,E1 -1360.165,E2 -1360.165} C_VEL
LIN {X 0,Y 587.504,Z 455.54,A -85,B 0,C 180,E1 -1361.209,E2 -1361.209} C_VEL
LIN {X 0,Y 587.577,Z 444.358,A -85,B 0,C 180,E1 -1362.083,E2 -1362.083} C_VEL
LIN {X 0,Y 587.635,Z 432.012,A -85,B 0,C 180,E1 -1362.871,E2 -1362.871} C_VEL
LIN {X 0,Y 587.759,Z 420.133,A -85,B 0,C 180,E1 -1363.484,E2 -1363.484} C_VEL
LIN {X 0,Y 587.879,Z 406.888,A -85,B 0,C 180,E1 -1364.019,E2 -1364.019} C_VEL
LIN {X 0,Y 587.933,Z 393.038,A -85,B 0,C 180,E1 -1364.433,E2 -1364.433} C_VEL
LIN {X 0,Y 587.791,Z 380.649,A -85,B 0,C 180,E1 -1364.69,E2 -1364.69} C_VEL
LIN {X 0,Y 587.21,Z 377.467,A -85,B 0,C 180,E1 -1364.756,E2 -1364.756} C_VEL
LIN {X 0,Y 587.21,Z 371.5,A -85,B 0,C 180,E1 -1367.41,E2 -1367.41} C_VEL
LIN {X 0,Y 587.208,Z 366.686,A -85,B 0,C 180,E1 -1369.58,E2 -1369.58} C_VEL
LIN {X 0,Y 587.217,Z 361.872,A -85,B 0,C 180,E1 -1371.779,E2 -1371.779} C_VEL
LIN {X 0,Y 587.246,Z 355.893,A -85,B 0,C 180,E1 -1374.557,E2 -1374.557} C_VEL
LIN {X 0,Y 587.241,Z 350.639,A -85,B 0,C 180,E1 -1377.051,E2 -1377.051} C_VEL
LIN {X 0,Y 587.289,Z 345.87,A -85,B 0,C 180,E1 -1379.383,E2 -1379.383} C_VEL
LIN {X 0,Y 587.349,Z 341.004,A -85,B 0,C 180,E1 -1381.836,E2 -1381.836} C_VEL
LIN {X 0,Y 587.364,Z 336.09,A -85,B 0,C 180,E1 -1384.35,E2 -1384.35} C_VEL
LIN {X 0,Y 587.407,Z 331.508,A -85,B 0,C 180,E1 -1386.743,E2 -1386.743} C_VEL
LIN {X 0,Y 587.357,Z 327.948,A -85,B 0,C 180,E1 -1388.65,E2 -1388.65} C_VEL
LIN {X 0,Y 587.341,Z 327.951,A -85,B 0,C 180,E1 -1391.157,E2 -1391.157} C_VEL
LIN {X 0,Y 587.332,Z 327.947,A -85,B 0,C 180,E1 -1394.114,E2 -1394.114} C_VEL
LIN {X 0,Y 587.318,Z 327.949,A -85,B 0,C 180,E1 -1396.994,E2 -1396.994} C_VEL
LIN {X 0,Y 587.319,Z 327.954,A -85,B 0,C 180,E1 -1399.746,E2 -1399.746} C_VEL
LIN {X 0,Y 587.349,Z 327.944,A -85,B 0,C 180,E1 -1402.392,E2 -1402.392} C_VEL
LIN {X 0,Y 587.367,Z 327.942,A -85,B 0,C 180,E1 -1405.78,E2 -1405.78} C_VEL
LIN {X 0,Y 587.343,Z 327.953,A -85,B 0,C 180,E1 -1408.231,E2 -1408.231} C_VEL
LIN {X 0,Y 587.356,Z 327.944,A -85,B 0,C 180,E1 -1410.867,E2 -1410.867} C_VEL
LIN {X 0,Y 587.342,Z 327.947,A -85,B 0,C 180,E1 -1413.721,E2 -1413.721} C_VEL
LIN {X 0,Y 587.341,Z 327.946,A -85,B 0,C 180,E1 -1415.994,E2 -1415.994} C_VEL
LIN {X 0,Y 587.327,Z 327.953,A -85,B 0,C 180,E1 -1418.226,E2 -1418.226} C_VEL
LIN {X 0,Y 587.352,Z 327.945,A -85,B 0,C 180,E1 -1421.151,E2 -1421.151} C_VEL
LIN {X 0,Y 587.33,Z 327.947,A -85,B 0,C 180,E1 -1424.025,E2 -1424.025} C_VEL
LIN {X 0,Y 587.357,Z 327.944,A -85,B 0,C 180,E1 -1426.154,E2 -1426.154} C_VEL
LIN {X 0,Y 587.344,Z 327.946,A -85,B 0,C 180,E1 -1428.962,E2 -1428.962} C_VEL
LIN {X 0,Y 587.346,Z 327.952,A -85,B 0,C 180,E1 -1431.744,E2 -1431.744} C_VEL
LIN {X 0,Y 587.362,Z 327.943,A -85,B 0,C 180,E1 -1434.507,E2 -1434.507} C_VEL
LIN {X 0,Y 587.379,Z 327.942,A -85,B 0,C 180,E1 -1437.257,E2 -1437.257} C_VEL
LIN {X 0,Y 587.387,Z 327.945,A -85,B 0,C 180,E1 -1440,E2 -1440} C_VEL
LIN {X 0,Y 587.377,Z 327.941,A -85,B 0,C 180,E1 -1442.743,E2 -1442.743} C_VEL
LIN {X 0,Y 587.363,Z 327.946,A -85,B 0,C 180,E1 -1445.493,E2 -1445.493} C_VEL
LIN {X 0,Y 587.347,Z 327.948,A -85,B 0,C 180,E1 -1448.255,E2 -1448.255} C_VEL
LIN {X 0,Y 587.355,Z 327.943,A -85,B 0,C 180,E1 -1451.133,E2 -1451.133} C_VEL
LIN {X 0,Y 587.372,Z 327.942,A -85,B 0,C 180,E1 -1454.26,E2 -1454.26} C_VEL
LIN {X 0,Y 587.355,Z 327.946,A -85,B 0,C 180,E1 -1457.406,E2 -1457.406} C_VEL
LIN {X 0,Y 587.319,Z 327.948,A -85,B 0,C 180,E1 -1459.576,E2 -1459.576} C_VEL
LIN {X 0,Y 587.344,Z 327.946,A -85,B 0,C 180,E1 -1462.514,E2 -1462.514} C_VEL
LIN {X 0,Y 587.357,Z 327.944,A -85,B 0,C 180,E1 -1464.758,E2 -1464.758} C_VEL
LIN {X 0,Y 587.357,Z 327.944,A -85,B 0,C 180,E1 -1467.693,E2 -1467.693} C_VEL
LIN {X 0,Y 587.342,Z 327.951,A -85,B 0,C 180,E1 -1470.51,E2 -1470.51} C_VEL
LIN {X 0,Y 587.337,Z 327.949,A -85,B 0,C 180,E1 -1473.396,E2 -1473.396} C_VEL
LIN {X 0,Y 587.354,Z 327.946,A -85,B 0,C 180,E1 -1475.896,E2 -1475.896} C_VEL
LIN {X 0,Y 587.333,Z 327.95,A -85,B 0,C 180,E1 -1478.479,E2 -1478.479} C_VEL
LIN {X 0,Y 587.339,Z 327.946,A -85,B 0,C 180,E1 -1481.157,E2 -1481.157} C_VEL
LIN {X 0,Y 587.315,Z 327.952,A -85,B 0,C 180,E1 -1484.112,E2 -1484.112} C_VEL
LIN {X 0,Y 587.327,Z 327.953,A -85,B 0,C 180,E1 -1486.994,E2 -1486.994} C_VEL
LIN {X 0,Y 587.316,Z 327.95,A -85,B 0,C 180,E1 -1489.745,E2 -1489.745} C_VEL
LIN {X 0,Y 587.348,Z 327.951,A -85,B 0,C 180,E1 -1492.392,E2 -1492.392} C_VEL
LIN {X 0,Y 587.352,Z 328.044,A -85,B 0,C 180,E1 -1494.26,E2 -1494.26} C_VEL
LIN {X 0,Y 587.876,Z 332.506,A -85,B 0,C 180,E1 -1495.577,E2 -1495.577} C_VEL
LIN {X 0,Y 587.752,Z 343.805,A -85,B 0,C 180,E1 -1498.657,E2 -1498.657} C_VEL
LIN {X 0,Y 587.634,Z 354.309,A -85,B 0,C 180,E1 -1501.419,E2 -1501.419} C_VEL
LIN {X 0,Y 587.539,Z 364.932,A -85,B 0,C 180,E1 -1504.135,E2 -1504.135} C_VEL
LIN {X 0,Y 587.484,Z 376.774,A -85,B 0,C 180,E1 -1507.093,E2 -1507.093} C_VEL
LIN {X 0,Y 587.391,Z 387.417,A -85,B 0,C 180,E1 -1509.697,E2 -1509.697} C_VEL
LIN {X 0,Y 587.335,Z 399.456,A -85,B 0,C 180,E1 -1512.593,E2 -1512.593} C_VEL
LIN {X 0,Y 587.34,Z 400.29,A -85,B 0,C 180,E1 -1512.792,E2 -1512.792} C_VEL
LIN {X 0,Y 588.293,Z 404.76,A -85,B 0,C 180,E1 -1512.885,E2 -1512.885} C_VEL
LIN {X 0,Y 588.263,Z 420.034,A -85,B 0,C 180,E1 -1513.15,E2 -1513.15} C_VEL
LIN {X 0,Y 588.17,Z 435.289,A -85,B 0,C 180,E1 -1513.558,E2 -1513.558} C_VEL
LIN {X 0,Y 588.031,Z 449.789,A -85,B 0,C 180,E1 -1514.089,E2 -1514.089} C_VEL
LIN {X 0,Y 587.93,Z 463.863,A -85,B 0,C 180,E1 -1514.753,E2 -1514.753} C_VEL
LIN {X 0,Y 587.791,Z 477.33,A -85,B 0,C 180,E1 -1515.539,E2 -1515.539} C_VEL
LIN {X 0,Y 587.644,Z 489.854,A -85,B 0,C 180,E1 -1516.425,E2 -1516.425} C_VEL
LIN {X 0,Y 587.549,Z 501.274,A -85,B 0,C 180,E1 -1517.391,E2 -1517.391} C_VEL
LIN {X 0,Y 587.405,Z 511.927,A -85,B 0,C 180,E1 -1518.457,E2 -1518.457} C_VEL
LIN {X 0,Y 587.35,Z 522.02,A -85,B 0,C 180,E1 -1519.66,E2 -1519.66} C_VEL
LIN {X 0,Y 587.267,Z 530.533,A -85,B 0,C 180,E1 -1520.876,E2 -1520.876} C_VEL
LIN {X 0,Y 587.252,Z 537.612,A -85,B 0,C 180,E1 -1522.089,E2 -1522.089} C_VEL
LIN {X 0,Y 587.204,Z 543.929,A -85,B 0,C 180,E1 -1523.409,E2 -1523.409} C_VEL
LIN {X 0,Y 587.157,Z 549.323,A -85,B 0,C 180,E1 -1524.849,E2 -1524.849} C_VEL
LIN {X 0,Y 587.167,Z 552.289,A -85,B 0,C 180,E1 -1525.882,E2 -1525.882} C_VEL
LIN {X 0,Y 587.129,Z 555.186,A -85,B 0,C 180,E1 -1527.256,E2 -1527.256} C_VEL
LIN {X 0,Y 587.145,Z 556.912,A -85,B 0,C 180,E1 -1528.628,E2 -1528.628} C_VEL
LIN {X 0,Y 587.134,Z 557.5,A -85,B 0,C 180,E1 -1530,E2 -1530} C_VEL
LIN {X 0,Y 587.145,Z 556.912,A -85,B 0,C 180,E1 -1531.372,E2 -1531.372} C_VEL
LIN {X 0,Y 587.129,Z 555.186,A -85,B 0,C 180,E1 -1532.744,E2 -1532.744} C_VEL
LIN {X 0,Y 587.167,Z 552.288,A -85,B 0,C 180,E1 -1534.118,E2 -1534.118} C_VEL
LIN {X 0,Y 587.199,Z 548.162,A -85,B 0,C 180,E1 -1535.494,E2 -1535.494} C_VEL
LIN {X 0,Y 587.206,Z 542.703,A -85,B 0,C 180,E1 -1536.874,E2 -1536.874} C_VEL
LIN {X 0,Y 587.255,Z 535.75,A -85,B 0,C 180,E1 -1538.257,E2 -1538.257} C_VEL
LIN {X 0,Y 587.286,Z 527.09,A -85,B 0,C 180,E1 -1539.645,E2 -1539.645} C_VEL
LIN {X 0,Y 587.371,Z 517.876,A -85,B 0,C 180,E1 -1540.862,E2 -1540.862} C_VEL
LIN {X 0,Y 587.446,Z 508.508,A -85,B 0,C 180,E1 -1541.91,E2 -1541.91} C_VEL
LIN {X 0,Y 587.558,Z 497.387,A -85,B 0,C 180,E1 -1542.96,E2 -1542.96} C_VEL
LIN {X 0,Y 587.711,Z 484.817,A -85,B 0,C 180,E1 -1543.953,E2 -1543.953} C_VEL
LIN {X 0,Y 587.832,Z 471.78,A -85,B 0,C 180,E1 -1544.807,E2 -1544.807} C_VEL
LIN {X 0,Y 587.954,Z 458.604,A -85,B 0,C 180,E1 -1545.513,E2 -1545.513} C_VEL
LIN {X 0,Y 588.086,Z 444.179,A -85,B 0,C 180,E1 -1546.132,E2 -1546.132} C_VEL
LIN {X 0,Y 588.203,Z 429.25,A -85,B 0,C 180,E1 -1546.619,E2 -1546.619} C_VEL
LIN {X 0,Y 588.272,Z 413.903,A -85,B 0,C 180,E1 -1546.972,E2 -1546.972} C_VEL
LIN {X 0,Y 588.134,Z 404.009,A -85,B 0,C 180,E1 -1547.13,E2 -1547.13} C_VEL
LIN {X 0,Y 587.363,Z 400.287,A -85,B 0,C 180,E1 -1547.207,E2 -1547.207} C_VEL
LIN {X 0,Y 587.391,Z 387.417,A -85,B 0,C 180,E1 -1550.303,E2 -1550.303} C_VEL
LIN {X 0,Y 587.503,Z 375.378,A -85,B 0,C 180,E1 -1553.251,E2 -1553.251} C_VEL
LIN {X 0,Y 587.552,Z 363.339,A -85,B 0,C 180,E1 -1556.268,E2 -1556.268} C_VEL
LIN {X 0,Y 587.658,Z 351.972,A -85,B 0,C 180,E1 -1559.187,E2 -1559.187} C_VEL
LIN {X 0,Y 587.767,Z 341.731,A -85,B 0,C 180,E1 -1561.902,E2 -1561.902} C_VEL
LIN {X 0,Y 587.869,Z 331.624,A -85,B 0,C 180,E1 -1564.675,E2 -1564.675} C_VEL
LIN {X 0,Y 587.321,Z 327.955,A -85,B 0,C 180,E1 -1565.794,E2 -1565.794} C_VEL
LIN {X 0,Y 587.331,Z 327.949,A -85,B 0,C 180,E1 -1568.48,E2 -1568.48} C_VEL
LIN {X 0,Y 587.339,Z 327.952,A -85,B 0,C 180,E1 -1571.157,E2 -1571.157} C_VEL
LIN {X 0,Y 587.337,Z 327.947,A -85,B 0,C 180,E1 -1574.114,E2 -1574.114} C_VEL
LIN {X 0,Y 587.315,Z 327.949,A -85,B 0,C 180,E1 -1576.994,E2 -1576.994} C_VEL
LIN {X 0,Y 587.322,Z 327.953,A -85,B 0,C 180,E1 -1579.746,E2 -1579.746} C_VEL
LIN {X 0,Y 587.348,Z 327.946,A -85,B 0,C 180,E1 -1582.393,E2 -1582.393} C_VEL
LIN {X 0,Y 587.353,Z 327.947,A -85,B 0,C 180,E1 -1584.946,E2 -1584.946} C_VEL
LIN {X 0,Y 587.337,Z 327.947,A -85,B 0,C 180,E1 -1587.421,E2 -1587.421} C_VEL
LIN {X 0,Y 587.337,Z 327.951,A -85,B 0,C 180,E1 -1589.83,E2 -1589.83} C_VEL
LIN {X 0,Y 587.355,Z 327.944,A -85,B 0,C 180,E1 -1592.307,E2 -1592.307} C_VEL
LIN {X 0,Y 587.356,Z 327.944,A -85,B 0,C 180,E1 -1595.242,E2 -1595.242} C_VEL
LIN {X 0,Y 587.322,Z 327.952,A -85,B 0,C 180,E1 -1598.226,E2 -1598.226} C_VEL
LIN {X 0,Y 587.356,Z 327.947,A -85,B 0,C 180,E1 -1601.152,E2 -1601.152} C_VEL
LIN {X 0,Y 587.326,Z 327.947,A -85,B 0,C 180,E1 -1604.025,E2 -1604.025} C_VEL
LIN {X 0,Y 587.365,Z 327.946,A -85,B 0,C 180,E1 -1606.155,E2 -1606.155} C_VEL
LIN {X 0,Y 587.343,Z 327.945,A -85,B 0,C 180,E1 -1608.963,E2 -1608.963} C_VEL
LIN {X 0,Y 587.346,Z 327.949,A -85,B 0,C 180,E1 -1611.745,E2 -1611.745} C_VEL
LIN {X 0,Y 587.363,Z 327.945,A -85,B 0,C 180,E1 -1614.507,E2 -1614.507} C_VEL
LIN {X 0,Y 587.377,Z 327.94,A -85,B 0,C 180,E1 -1617.257,E2 -1617.257} C_VEL
LIN {X 0,Y 587.389,Z 327.945,A -85,B 0,C 180,E1 -1620,E2 -1620} C_VEL
LIN {X 0,Y 587.378,Z 327.942,A -85,B 0,C 180,E1 -1622.743,E2 -1622.743} C_VEL
LIN {X 0,Y 587.362,Z 327.944,A -85,B 0,C 180,E1 -1625.493,E2 -1625.493} C_VEL
LIN {X 0,Y 587.346,Z 327.951,A -85,B 0,C 180,E1 -1628.256,E2 -1628.256} C_VEL
LIN {X 0,Y 587.354,Z 327.944,A -85,B 0,C 180,E1 -1631.134,E2 -1631.134} C_VEL
LIN {X 0,Y 587.37,Z 327.942,A -85,B 0,C 180,E1 -1634.26,E2 -1634.26} C_VEL
LIN {X 0,Y 587.355,Z 327.944,A -85,B 0,C 180,E1 -1637.406,E2 -1637.406} C_VEL
LIN {X 0,Y 587.314,Z 327.951,A -85,B 0,C 180,E1 -1638.314,E2 -1638.314} C_VEL
LIN {X 0,Y 586.672,Z 328.031,A -85,B 0,C 180,E1 -1638.886,E2 -1638.886} C_VEL
LIN {X 0,Y 583.848,Z 328.384,A -85,B 0,C 180,E1 -1639.814,E2 -1639.814} C_VEL
LIN {X 0,Y 581.437,Z 328.685,A -85,B 0,C 180,E1 -1640.561,E2 -1640.561} C_VEL
LIN {X 0,Y 580.383,Z 328.814,A -85,B 0,C 180,E1 -1641.138,E2 -1641.138} C_VEL
LIN {X 0,Y 580.288,Z 328.825,A -85,B 0,C 180,E1 -1641.333,E2 -1641.333} C_VEL
LIN {X 0,Y 580.306,Z 328.821,A -85,B 0,C 180,E1 -1644.316,E2 -1644.316} C_VEL
LIN {X 0,Y 580.293,Z 328.824,A -85,B 0,C 180,E1 -1647.402,E2 -1647.402} C_VEL
LIN {X 0,Y 580.293,Z 328.825,A -85,B 0,C 180,E1 -1649.773,E2 -1649.773} C_VEL
LIN {X 0,Y 580.301,Z 328.825,A -85,B 0,C 180,E1 -1652.201,E2 -1652.201} C_VEL
LIN {X 0,Y 580.295,Z 328.824,A -85,B 0,C 180,E1 -1654.696,E2 -1654.696} C_VEL
LIN {X 0,Y 580.302,Z 328.825,A -85,B 0,C 180,E1 -1657.268,E2 -1657.268} C_VEL
LIN {X 0,Y 580.297,Z 328.83,A -85,B 0,C 180,E1 -1660.271,E2 -1660.271} C_VEL
LIN {X 0,Y 580.281,Z 328.825,A -85,B 0,C 180,E1 -1662.706,E2 -1662.706} C_VEL
LIN {X 0,Y 580.274,Z 328.829,A -85,B 0,C 180,E1 -1665.609,E2 -1665.609} C_VEL
LIN {X 0,Y 580.318,Z 328.823,A -85,B 0,C 180,E1 -1668.234,E2 -1668.234} C_VEL
LIN {X 0,Y 580.324,Z 328.823,A -85,B 0,C 180,E1 -1671.358,E2 -1671.358} C_VEL
LIN {X 0,Y 580.385,Z 334.187,A -85,B 0,C 180,E1 -1674.225,E2 -1674.225} C_VEL
LIN {X 0,Y 580.302,Z 339.417,A -85,B 0,C 180,E1 -1676.976,E2 -1676.976} C_VEL
LIN {X 0,Y 580.284,Z 344.178,A -85,B 0,C 180,E1 -1679.424,E2 -1679.424} C_VEL
LIN {X 0,Y 580.224,Z 349.615,A -85,B 0,C 180,E1 -1682.156,E2 -1682.156} C_VEL
LIN {X 0,Y 580.182,Z 355.264,A -85,B 0,C 180,E1 -1684.914,E2 -1684.914} C_VEL
LIN {X 0,Y 580.173,Z 360.075,A -85,B 0,C 180,E1 -1687.192,E2 -1687.192} C_VEL
LIN {X 0,Y 580.122,Z 364.886,A -85,B 0,C 180,E1 -1689.431,E2 -1689.431} C_VEL
LIN {X 0,Y 580.127,Z 369.697,A -85,B 0,C 180,E1 -1691.64,E2 -1691.64} C_VEL
LIN {X 0,Y 580.117,Z 374.508,A -85,B 0,C 180,E1 -1693.821,E2 -1693.821} C_VEL
LIN {X 0,Y 580.131,Z 377.465,A -85,B 0,C 180,E1 -1695.149,E2 -1695.149} C_VEL
LIN {X 0,Y 581.13,Z 384.013,A -85,B 0,C 180,E1 -1695.288,E2 -1695.288} C_VEL
LIN {X 0,Y 581.005,Z 398.421,A -85,B 0,C 180,E1 -1695.628,E2 -1695.628} C_VEL
LIN {X 0,Y 580.902,Z 412.947,A -85,B 0,C 180,E1 -1696.131,E2 -1696.131} C_VEL
LIN {X 0,Y 580.772,Z 425.502,A -85,B 0,C 180,E1 -1696.708,E2 -1696.708} C_VEL
LIN {X 0,Y 580.658,Z 437.795,A -85,B 0,C 180,E1 -1697.416,E2 -1697.416} C_VEL
LIN {X 0,Y 580.54,Z 450.204,A -85,B 0,C 180,E1 -1698.301,E2 -1698.301} C_VEL
LIN {X 0,Y 580.442,Z 460.393,A -85,B 0,C 180,E1 -1699.185,E2 -1699.185} C_VEL
LIN {X 0,Y 580.28,Z 470.47,A -85,B 0,C 180,E1 -1700.238,E2 -1700.238} C_VEL
LIN {X 0,Y 580.241,Z 478.853,A -85,B 0,C 180,E1 -1701.292,E2 -1701.292} C_VEL
LIN {X 0,Y 580.166,Z 486.865,A -85,B 0,C 180,E1 -1702.518,E2 -1702.518} C_VEL
LIN {X 0,Y 580.104,Z 493.318,A -85,B 0,C 180,E1 -1703.74,E2 -1703.74} C_VEL
LIN {X 0,Y 580.077,Z 497.797,A -85,B 0,C 180,E1 -1704.787,E2 -1704.787} C_VEL
LIN {X 0,Y 580.103,Z 501.306,A -85,B 0,C 180,E1 -1705.832,E2 -1705.832} C_VEL
LIN {X 0,Y 580.041,Z 504.739,A -85,B 0,C 180,E1 -1707.222,E2 -1707.222} C_VEL
LIN {X 0,Y 580.045,Z 506.782,A -85,B 0,C 180,E1 -1708.611,E2 -1708.611} C_VEL
LIN {X 0,Y 580.037,Z 507.496,A -85,B 0,C 180,E1 -1710,E2 -1710} C_VEL
LIN {X 0,Y 580.042,Z 506.882,A -85,B 0,C 180,E1 -1711.389,E2 -1711.389} C_VEL
LIN {X 0,Y 580.039,Z 504.926,A -85,B 0,C 180,E1 -1712.778,E2 -1712.778} C_VEL
LIN {X 0,Y 580.104,Z 501.579,A -85,B 0,C 180,E1 -1714.169,E2 -1714.169} C_VEL
LIN {X 0,Y 580.129,Z 496.75,A -85,B 0,C 180,E1 -1715.562,E2 -1715.562} C_VEL
LIN {X 0,Y 580.142,Z 490.286,A -85,B 0,C 180,E1 -1716.958,E2 -1716.958} C_VEL
LIN {X 0,Y 580.193,Z 483.086,A -85,B 0,C 180,E1 -1718.183,E2 -1718.183} C_VEL
LIN {X 0,Y 580.284,Z 475.547,A -85,B 0,C 180,E1 -1719.235,E2 -1719.235} C_VEL
LIN {X 0,Y 580.347,Z 466.495,A -85,B 0,C 180,E1 -1720.29,E2 -1720.29} C_VEL
LIN {X 0,Y 580.495,Z 455.534,A -85,B 0,C 180,E1 -1721.346,E2 -1721.346} C_VEL
LIN {X 0,Y 580.583,Z 444.352,A -85,B 0,C 180,E1 -1722.23,E2 -1722.23} C_VEL
LIN {X 0,Y 580.695,Z 432.004,A -85,B 0,C 180,E1 -1723.027,E2 -1723.027} C_VEL
LIN {X 0,Y 580.85,Z 420.123,A -85,B 0,C 180,E1 -1723.647,E2 -1723.647} C_VEL
LIN {X 0,Y 580.986,Z 407.252,A -85,B 0,C 180,E1 -1724.176,E2 -1724.176} C_VEL
LIN {X 0,Y 581.061,Z 393.116,A -85,B 0,C 180,E1 -1724.605,E2 -1724.605} C_VEL
LIN {X 0,Y 580.926,Z 381.664,A -85,B 0,C 180,E1 -1724.852,E2 -1724.852} C_VEL
LIN {X 0,Y 580.115,Z 377.465,A -85,B 0,C 180,E1 -1724.941,E2 -1724.941} C_VEL
LIN {X 0,Y 580.12,Z 371.499,A -85,B 0,C 180,E1 -1727.63,E2 -1727.63} C_VEL
LIN {X 0,Y 580.118,Z 366.685,A -85,B 0,C 180,E1 -1729.829,E2 -1729.829} C_VEL
LIN {X 0,Y 580.153,Z 361.871,A -85,B 0,C 180,E1 -1732.058,E2 -1732.058} C_VEL
LIN {X 0,Y 580.182,Z 355.452,A -85,B 0,C 180,E1 -1735.086,E2 -1735.086} C_VEL
LIN {X 0,Y 580.225,Z 349.802,A -85,B 0,C 180,E1 -1737.845,E2 -1737.845} C_VEL
LIN {X 0,Y 580.261,Z 344.149,A -85,B 0,C 180,E1 -1740.69,E2 -1740.69} C_VEL
LIN {X 0,Y 580.33,Z 339.025,A -85,B 0,C 180,E1 -1743.32,E2 -1743.32} C_VEL
LIN {X 0,Y 580.375,Z 333.18,A -85,B 0,C 180,E1 -1746.396,E2 -1746.396} C_VEL
LIN {X 0,Y 580.318,Z 328.826,A -85,B 0,C 180,E1 -1748.698,E2 -1748.698} C_VEL
LIN {X 0,Y 580.283,Z 328.833,A -85,B 0,C 180,E1 -1751.331,E2 -1751.331} C_VEL
LIN {X 0,Y 580.284,Z 328.826,A -85,B 0,C 180,E1 -1753.658,E2 -1753.658} C_VEL
LIN {X 0,Y 580.279,Z 328.83,A -85,B 0,C 180,E1 -1756.61,E2 -1756.61} C_VEL
LIN {X 0,Y 580.303,Z 328.822,A -85,B 0,C 180,E1 -1759.157,E2 -1759.157} C_VEL
LIN {X 0,Y 580.295,Z 328.825,A -85,B 0,C 180,E1 -1761.927,E2 -1761.927} C_VEL
LIN {X 0,Y 580.258,Z 328.83,A -85,B 0,C 180,E1 -1764.453,E2 -1764.453} C_VEL
LIN {X 0,Y 580.295,Z 328.825,A -85,B 0,C 180,E1 -1766.975,E2 -1766.975} C_VEL
LIN {X 0,Y 580.302,Z 328.824,A -85,B 0,C 180,E1 -1769.425,E2 -1769.425} C_VEL
LIN {X 0,Y 580.305,Z 328.823,A -85,B 0,C 180,E1 -1772.141,E2 -1772.141} C_VEL
LIN {X 0,Y 580.328,Z 328.822,A -85,B 0,C 180,E1 -1775.27,E2 -1775.27} C_VEL
LIN {X 0,Y 580.277,Z 328.828,A -85,B 0,C 180,E1 -1777.947,E2 -1777.947} C_VEL
LIN {X 0,Y 580.303,Z 328.822,A -85,B 0,C 180,E1 -1780.913,E2 -1780.913} C_VEL
LIN {X 0,Y 580.285,Z 328.826,A -85,B 0,C 180,E1 -1783.826,E2 -1783.826} C_VEL
LIN {X 0,Y 580.324,Z 328.819,A -85,B 0,C 180,E1 -1785.983,E2 -1785.983} C_VEL
LIN {X 0,Y 580.312,Z 328.823,A -85,B 0,C 180,E1 -1788.827,E2 -1788.827} C_VEL
LIN {X 0,Y 580.316,Z 328.826,A -85,B 0,C 180,E1 -1791.644,E2 -1791.644} C_VEL
LIN {X 0,Y 580.285,Z 328.827,A -85,B 0,C 180,E1 -1793.742,E2 -1793.742} C_VEL
LIN {X 0,Y 580.268,Z 328.826,A -85,B 0,C 180,E1 -1795.833,E2 -1795.833} C_VEL
LIN {X 0,Y 580.335,Z 328.819,A -85,B 0,C 180,E1 -1797.918,E2 -1797.918} C_VEL
LIN {X 0,Y 580.366,Z 328.815,A -85,B 0,C 180,E1 -1800.694,E2 -1800.694} C_VEL
LIN {X 0,Y 580.284,Z 328.832,A -85,B 0,C 180,E1 -1803.472,E2 -1803.472} C_VEL
LIN {X 0,Y 580.328,Z 328.821,A -85,B 0,C 180,E1 -1805.56,E2 -1805.56} C_VEL
LIN {X 0,Y 580.33,Z 328.818,A -85,B 0,C 180,E1 -1807.655,E2 -1807.655} C_VEL
LIN {X 0,Y 580.301,Z 328.826,A -85,B 0,C 180,E1 -1810.467,E2 -1810.467} C_VEL
LIN {X 0,Y 580.31,Z 328.822,A -85,B 0,C 180,E1 -1812.591,E2 -1812.591} C_VEL
LIN {X 0,Y 580.292,Z 328.825,A -85,B 0,C 180,E1 -1814.734,E2 -1814.734} C_VEL
LIN {X 0,Y 580.299,Z 328.823,A -85,B 0,C 180,E1 -1817.624,E2 -1817.624} C_VEL
LIN {X 0,Y 580.293,Z 328.825,A -85,B 0,C 180,E1 -1819.823,E2 -1819.823} C_VEL
LIN {X 0,Y 580.275,Z 328.832,A -85,B 0,C 180,E1 -1822.052,E2 -1822.052} C_VEL
LIN {X 0,Y 580.312,Z 328.825,A -85,B 0,C 180,E1 -1825.079,E2 -1825.079} C_VEL
LIN {X 0,Y 580.304,Z 328.823,A -85,B 0,C 180,E1 -1828.185,E2 -1828.185} C_VEL
LIN {X 0,Y 580.289,Z 328.827,A -85,B 0,C 180,E1 -1830.694,E2 -1830.694} C_VEL
LIN {X 0,Y 580.306,Z 328.824,A -85,B 0,C 180,E1 -1833.316,E2 -1833.316} C_VEL
LIN {X 0,Y 580.326,Z 328.823,A -85,B 0,C 180,E1 -1835.766,E2 -1835.766} C_VEL
LIN {X 0,Y 580.292,Z 328.824,A -85,B 0,C 180,E1 -1838.146,E2 -1838.146} C_VEL
LIN {X 0,Y 580.302,Z 328.825,A -85,B 0,C 180,E1 -1840.843,E2 -1840.843} C_VEL
LIN {X 0,Y 580.276,Z 328.832,A -85,B 0,C 180,E1 -1843.658,E2 -1843.658} C_VEL
LIN {X 0,Y 580.29,Z 328.826,A -85,B 0,C 180,E1 -1846.608,E2 -1846.608} C_VEL
LIN {X 0,Y 580.302,Z 328.827,A -85,B 0,C 180,E1 -1849.156,E2 -1849.156} C_VEL
LIN {X 0,Y 580.293,Z 328.828,A -85,B 0,C 180,E1 -1851.927,E2 -1851.927} C_VEL
LIN {X 0,Y 580.321,Z 328.88,A -85,B 0,C 180,E1 -1853.998,E2 -1853.998} C_VEL
LIN {X 0,Y 580.95,Z 333.363,A -85,B 0,C 180,E1 -1855.348,E2 -1855.348} C_VEL
LIN {X 0,Y 580.84,Z 342.48,A -85,B 0,C 180,E1 -1857.885,E2 -1857.885} C_VEL
LIN {X 0,Y 580.719,Z 352.679,A -85,B 0,C 180,E1 -1860.617,E2 -1860.617} C_VEL
LIN {X 0,Y 580.569,Z 364.194,A -85,B 0,C 180,E1 -1863.611,E2 -1863.611} C_VEL
LIN {X 0,Y 580.485,Z 375.378,A -85,B 0,C 180,E1 -1866.451,E2 -1866.451} C_VEL
LIN {X 0,Y 580.367,Z 387.417,A -85,B 0,C 180,E1 -1869.44,E2 -1869.44} C_VEL
LIN {X 0,Y 580.299,Z 399.456,A -85,B 0,C 180,E1 -1872.375,E2 -1872.375} C_VEL
LIN {X 0,Y 580.306,Z 400.286,A -85,B 0,C 180,E1 -1872.576,E2 -1872.576} C_VEL
LIN {X 0,Y 581.527,Z 405.961,A -85,B 0,C 180,E1 -1872.697,E2 -1872.697} C_VEL
LIN {X 0,Y 581.457,Z 420.866,A -85,B 0,C 180,E1 -1872.967,E2 -1872.967} C_VEL
LIN {X 0,Y 581.354,Z 435.288,A -85,B 0,C 180,E1 -1873.36,E2 -1873.36} C_VEL
LIN {X 0,Y 581.181,Z 449.791,A -85,B 0,C 180,E1 -1873.896,E2 -1873.896} C_VEL
LIN {X 0,Y 581.04,Z 463.866,A -85,B 0,C 180,E1 -1874.567,E2 -1874.567} C_VEL
LIN {X 0,Y 580.872,Z 477.556,A -85,B 0,C 180,E1 -1875.377,E2 -1875.377} C_VEL
LIN {X 0,Y 580.677,Z 491.012,A -85,B 0,C 180,E1 -1876.349,E2 -1876.349} C_VEL
LIN {X 0,Y 580.541,Z 503.188,A -85,B 0,C 180,E1 -1877.414,E2 -1877.414} C_VEL
LIN {X 0,Y 580.385,Z 513.704,A -85,B 0,C 180,E1 -1878.51,E2 -1878.51} C_VEL
LIN {X 0,Y 580.309,Z 523.369,A -85,B 0,C 180,E1 -1879.71,E2 -1879.71} C_VEL
LIN {X 0,Y 580.207,Z 531.651,A -85,B 0,C 180,E1 -1880.94,E2 -1880.94} C_VEL
LIN {X 0,Y 580.165,Z 539.424,A -85,B 0,C 180,E1 -1882.342,E2 -1882.342} C_VEL
LIN {X 0,Y 580.094,Z 545.606,A -85,B 0,C 180,E1 -1883.74,E2 -1883.74} C_VEL
LIN {X 0,Y 580.041,Z 550.384,A -85,B 0,C 180,E1 -1885.135,E2 -1885.135} C_VEL
LIN {X 0,Y 580.104,Z 553.888,A -85,B 0,C 180,E1 -1886.527,E2 -1886.527} C_VEL
LIN {X 0,Y 580.039,Z 556.193,A -85,B 0,C 180,E1 -1887.917,E2 -1887.917} C_VEL
LIN {X 0,Y 580.038,Z 557.35,A -85,B 0,C 180,E1 -1889.306,E2 -1889.306} C_VEL
LIN {X 0,Y 580.038,Z 557.349,A -85,B 0,C 180,E1 -1890.694,E2 -1890.694} C_VEL
LIN {X 0,Y 580.039,Z 556.192,A -85,B 0,C 180,E1 -1892.083,E2 -1892.083} C_VEL
LIN {X 0,Y 580.104,Z 553.886,A -85,B 0,C 180,E1 -1893.473,E2 -1893.473} C_VEL
LIN {X 0,Y 580.041,Z 550.384,A -85,B 0,C 180,E1 -1894.865,E2 -1894.865} C_VEL
LIN {X 0,Y 580.093,Z 545.608,A -85,B 0,C 180,E1 -1896.26,E2 -1896.26} C_VEL
LIN {X 0,Y 580.165,Z 539.424,A -85,B 0,C 180,E1 -1897.658,E2 -1897.658} C_VEL
LIN {X 0,Y 580.207,Z 531.65,A -85,B 0,C 180,E1 -1899.06,E2 -1899.06} C_VEL
LIN {X 0,Y 580.309,Z 523.369,A -85,B 0,C 180,E1 -1900.29,E2 -1900.29} C_VEL
LIN {X 0,Y 580.383,Z 513.394,A -85,B 0,C 180,E1 -1901.525,E2 -1901.525} C_VEL
LIN {X 0,Y 580.541,Z 503.19,A -85,B 0,C 180,E1 -1902.586,E2 -1902.586} C_VEL
LIN {X 0,Y 580.678,Z 491.017,A -85,B 0,C 180,E1 -1903.651,E2 -1903.651} C_VEL
LIN {X 0,Y 580.846,Z 478.805,A -85,B 0,C 180,E1 -1904.542,E2 -1904.542} C_VEL
LIN {X 0,Y 580.996,Z 465.519,A -85,B 0,C 180,E1 -1905.344,E2 -1905.344} C_VEL
LIN {X 0,Y 581.153,Z 450.834,A -85,B 0,C 180,E1 -1906.059,E2 -1906.059} C_VEL
LIN {X 0,Y 581.347,Z 436.614,A -85,B 0,C 180,E1 -1906.595,E2 -1906.595} C_VEL
LIN {X 0,Y 581.445,Z 421.563,A -85,B 0,C 180,E1 -1907.017,E2 -1907.017} C_VEL
LIN {X 0,Y 581.497,Z 406.656,A -85,B 0,C 180,E1 -1907.293,E2 -1907.293} C_VEL
LIN {X 0,Y 580.336,Z 400.282,A -85,B 0,C 180,E1 -1907.424,E2 -1907.424} C_VEL
LIN {X 0,Y 580.357,Z 388.922,A -85,B 0,C 180,E1 -1910.19,E2 -1910.19} C_VEL
LIN {X 0,Y 580.479,Z 377.36,A -85,B 0,C 180,E1 -1913.052,E2 -1913.052} C_VEL
LIN {X 0,Y 580.579,Z 365.271,A -85,B 0,C 180,E1 -1916.112,E2 -1916.112} C_VEL
LIN {X 0,Y 580.663,Z 354.31,A -85,B 0,C 180,E1 -1918.956,E2 -1918.956} C_VEL
LIN {X 0,Y 580.822,Z 343.875,A -85,B 0,C 180,E1 -1921.734,E2 -1921.734} C_VEL
LIN {X 0,Y 580.925,Z 334.851,A -85,B 0,C 180,E1 -1924.233,E2 -1924.233} C_VEL
LIN {X 0,Y 580.859,Z 331.891,A -85,B 0,C 180,E1 -1925.08,E2 -1925.08} C_VEL
LIN {X 0,Y 580.298,Z 328.83,A -85,B 0,C 180,E1 -1926.051,E2 -1926.051} C_VEL
LIN {X 0,Y 580.28,Z 328.829,A -85,B 0,C 180,E1 -1929.035,E2 -1929.035} C_VEL
LIN {X 0,Y 580.316,Z 328.821,A -85,B 0,C 180,E1 -1931.766,E2 -1931.766} C_VEL
LIN {X 0,Y 580.265,Z 328.833,A -85,B 0,C 180,E1 -1934.627,E2 -1934.627} C_VEL
LIN {X 0,Y 580.288,Z 328.829,A -85,B 0,C 180,E1 -1937.628,E2 -1937.628} C_VEL
LIN {X 0,Y 580.298,Z 328.824,A -85,B 0,C 180,E1 -1940.068,E2 -1940.068} C_VEL
LIN {X 0,Y 580.306,Z 328.828,A -85,B 0,C 180,E1 -1943.065,E2 -1943.065} C_VEL
LIN {X 0,Y 580.306,Z 328.822,A -85,B 0,C 180,E1 -1945.441,E2 -1945.441} C_VEL
LIN {X 0,Y 580.303,Z 328.83,A -85,B 0,C 180,E1 -1947.97,E2 -1947.97} C_VEL
LIN {X 0,Y 580.306,Z 328.823,A -85,B 0,C 180,E1 -1950.69,E2 -1950.69} C_VEL
LIN {X 0,Y 580.295,Z 328.824,A -85,B 0,C 180,E1 -1953.666,E2 -1953.666} C_VEL
LIN {X 0,Y 580.306,Z 328.822,A -85,B 0,C 180,E1 -1955.684,E2 -1955.684} C_VEL
LIN {X 0,Y 580.274,Z 328.832,A -85,B 0,C 180,E1 -1957.948,E2 -1957.948} C_VEL
LIN {X 0,Y 580.305,Z 328.823,A -85,B 0,C 180,E1 -1960.914,E2 -1960.914} C_VEL
LIN {X 0,Y 580.282,Z 328.824,A -85,B 0,C 180,E1 -1963.826,E2 -1963.826} C_VEL
LIN {X 0,Y 580.332,Z 328.82,A -85,B 0,C 180,E1 -1965.983,E2 -1965.983} C_VEL
LIN {X 0,Y 580.31,Z 328.821,A -85,B 0,C 180,E1 -1968.827,E2 -1968.827} C_VEL
LIN {X 0,Y 580.315,Z 328.826,A -85,B 0,C 180,E1 -1971.644,E2 -1971.644} C_VEL
LIN {X 0,Y 580.284,Z 328.825,A -85,B 0,C 180,E1 -1973.742,E2 -1973.742} C_VEL
LIN {X 0,Y 580.268,Z 328.827,A -85,B 0,C 180,E1 -1975.833,E2 -1975.833} C_VEL
LIN {X 0,Y 580.343,Z 328.82,A -85,B 0,C 180,E1 -1977.918,E2 -1977.918} C_VEL
LIN {X 0,Y 580.365,Z 328.814,A -85,B 0,C 180,E1 -1980.694,E2 -1980.694} C_VEL
LIN {X 0,Y 580.285,Z 328.828,A -85,B 0,C 180,E1 -1983.472,E2 -1983.472} C_VEL
LIN {X 0,Y 580.328,Z 328.82,A -85,B 0,C 180,E1 -1985.56,E2 -1985.56} C_VEL
LIN {X 0,Y 580.328,Z 328.819,A -85,B 0,C 180,E1 -1987.656,E2 -1987.656} C_VEL
LIN {X 0,Y 580.304,Z 328.823,A -85,B 0,C 180,E1 -1990.467,E2 -1990.467} C_VEL
LIN {X 0,Y 580.309,Z 328.821,A -85,B 0,C 180,E1 -1992.591,E2 -1992.591} C_VEL
LIN {X 0,Y 580.292,Z 328.826,A -85,B 0,C 180,E1 -1994.734,E2 -1994.734} C_VEL
LIN {X 0,Y 580.298,Z 328.822,A -85,B 0,C 180,E1 -1997.625,E2 -1997.625} C_VEL
LIN {X 0,Y 580.292,Z 328.827,A -85,B 0,C 180,E1 -1999.823,E2 -1999.823} C_VEL
LIN {X 0,Y 580.288,Z 328.825,A -85,B 0,C 180,E1 -2001.333,E2 -2001.333} C_VEL
LIN {X 0,Y 579.59,Z 328.916,A -85,B 0,C 180,E1 -2001.912,E2 -2001.912} C_VEL
LIN {X 0,Y 576.714,Z 329.27,A -85,B 0,C 180,E1 -2002.852,E2 -2002.852} C_VEL
LIN {X 0,Y 574.32,Z 329.572,A -85,B 0,C 180,E1 -2003.608,E2 -2003.608} C_VEL
LIN {X 0,Y 573.322,Z 329.692,A -85,B 0,C 180,E1 -2004.192,E2 -2004.192} C_VEL
LIN {X 0,Y 573.255,Z 329.699,A -85,B 0,C 180,E1 -2004.389,E2 -2004.389} C_VEL
LIN {X 0,Y 573.255,Z 329.705,A -85,B 0,C 180,E1 -2006.976,E2 -2006.976} C_VEL
LIN {X 0,Y 573.252,Z 329.7,A -85,B 0,C 180,E1 -2009.488,E2 -2009.488} C_VEL
LIN {X 0,Y 573.257,Z 329.7,A -85,B 0,C 180,E1 -2012.645,E2 -2012.645} C_VEL
LIN {X 0,Y 573.213,Z 329.713,A -85,B 0,C 180,E1 -2015.188,E2 -2015.188} C_VEL
LIN {X 0,Y 573.239,Z 329.702,A -85,B 0,C 180,E1 -2017.808,E2 -2017.808} C_VEL
LIN {X 0,Y 573.249,Z 329.705,A -85,B 0,C 180,E1 -2020.525,E2 -2020.525} C_VEL
LIN {X 0,Y 573.243,Z 329.706,A -85,B 0,C 180,E1 -2023.359,E2 -2023.359} C_VEL
LIN {X 0,Y 573.249,Z 329.702,A -85,B 0,C 180,E1 -2026.331,E2 -2026.331} C_VEL
LIN {X 0,Y 573.248,Z 329.708,A -85,B 0,C 180,E1 -2028.544,E2 -2028.544} C_VEL
LIN {X 0,Y 573.308,Z 329.904,A -85,B 0,C 180,E1 -2031.413,E2 -2031.413} C_VEL
LIN {X 0,Y 573.356,Z 334.763,A -85,B 0,C 180,E1 -2033.999,E2 -2033.999} C_VEL
LIN {X 0,Y 573.289,Z 339.499,A -85,B 0,C 180,E1 -2036.519,E2 -2036.519} C_VEL
LIN {X 0,Y 573.22,Z 344.469,A -85,B 0,C 180,E1 -2039.12,E2 -2039.12} C_VEL
LIN {X 0,Y 573.183,Z 350.092,A -85,B 0,C 180,E1 -2041.984,E2 -2041.984} C_VEL
LIN {X 0,Y 573.118,Z 355.28,A -85,B 0,C 180,E1 -2044.583,E2 -2044.583} C_VEL
LIN {X 0,Y 573.075,Z 361.68,A -85,B 0,C 180,E1 -2047.655,E2 -2047.655} C_VEL
LIN {X 0,Y 573.028,Z 366.491,A -85,B 0,C 180,E1 -2049.915,E2 -2049.915} C_VEL
LIN {X 0,Y 573.057,Z 371.302,A -85,B 0,C 180,E1 -2052.145,E2 -2052.145} C_VEL
LIN {X 0,Y 573.041,Z 377.467,A -85,B 0,C 180,E1 -2054.961,E2 -2054.961} C_VEL
LIN {X 0,Y 574.262,Z 384.042,A -85,B 0,C 180,E1 -2055.108,E2 -2055.108} C_VEL
LIN {X 0,Y 574.135,Z 398.44,A -85,B 0,C 180,E1 -2055.453,E2 -2055.453} C_VEL
LIN {X 0,Y 574.004,Z 412.963,A -85,B 0,C 180,E1 -2055.961,E2 -2055.961} C_VEL
LIN {X 0,Y 573.868,Z 425.515,A -85,B 0,C 180,E1 -2056.545,E2 -2056.545} C_VEL
LIN {X 0,Y 573.683,Z 437.806,A -85,B 0,C 180,E1 -2057.261,E2 -2057.261} C_VEL
LIN {X 0,Y 573.551,Z 450.212,A -85,B 0,C 180,E1 -2058.156,E2 -2058.156} C_VEL
LIN {X 0,Y 573.438,Z 460.706,A -85,B 0,C 180,E1 -2059.081,E2 -2059.081} C_VEL
LIN {X 0,Y 573.245,Z 470.475,A -85,B 0,C 180,E1 -2060.117,E2 -2060.117} C_VEL
LIN {X 0,Y 573.202,Z 478.858,A -85,B 0,C 180,E1 -2061.184,E2 -2061.184} C_VEL
LIN {X 0,Y 573.111,Z 486.868,A -85,B 0,C 180,E1 -2062.425,E2 -2062.425} C_VEL
LIN {X 0,Y 573.022,Z 493.321,A -85,B 0,C 180,E1 -2063.663,E2 -2063.663} C_VEL
LIN {X 0,Y 573,Z 497.799,A -85,B 0,C 180,E1 -2064.722,E2 -2064.722} C_VEL
LIN {X 0,Y 573.029,Z 501.308,A -85,B 0,C 180,E1 -2065.78,E2 -2065.78} C_VEL
LIN {X 0,Y 572.957,Z 504.741,A -85,B 0,C 180,E1 -2067.188,E2 -2067.188} C_VEL
LIN {X 0,Y 572.944,Z 506.783,A -85,B 0,C 180,E1 -2068.594,E2 -2068.594} C_VEL
LIN {X 0,Y 572.937,Z 507.496,A -85,B 0,C 180,E1 -2070,E2 -2070} C_VEL
LIN {X 0,Y 572.942,Z 506.881,A -85,B 0,C 180,E1 -2071.406,E2 -2071.406} C_VEL
LIN {X 0,Y 572.954,Z 504.926,A -85,B 0,C 180,E1 -2072.812,E2 -2072.812} C_VEL
LIN {X 0,Y 573.03,Z 501.578,A -85,B 0,C 180,E1 -2074.22,E2 -2074.22} C_VEL
LIN {X 0,Y 573.056,Z 496.748,A -85,B 0,C 180,E1 -2075.631,E2 -2075.631} C_VEL
LIN {X 0,Y 573.054,Z 490.284,A -85,B 0,C 180,E1 -2077.045,E2 -2077.045} C_VEL
LIN {X 0,Y 573.142,Z 483.083,A -85,B 0,C 180,E1 -2078.284,E2 -2078.284} C_VEL
LIN {X 0,Y 573.225,Z 474.181,A -85,B 0,C 180,E1 -2079.527,E2 -2079.527} C_VEL
LIN {X 0,Y 573.351,Z 464.837,A -85,B 0,C 180,E1 -2080.595,E2 -2080.595} C_VEL
LIN {X 0,Y 573.477,Z 454.481,A -85,B 0,C 180,E1 -2081.576,E2 -2081.576} C_VEL
LIN {X 0,Y 573.628,Z 443.067,A -85,B 0,C 180,E1 -2082.471,E2 -2082.471} C_VEL
LIN {X 0,Y 573.793,Z 430.43,A -85,B 0,C 180,E1 -2083.277,E2 -2083.277} C_VEL
LIN {X 0,Y 573.953,Z 418.143,A -85,B 0,C 180,E1 -2083.905,E2 -2083.905} C_VEL
LIN {X 0,Y 574.13,Z 404.491,A -85,B 0,C 180,E1 -2084.445,E2 -2084.445} C_VEL
LIN {X 0,Y 574.209,Z 390.381,A -85,B 0,C 180,E1 -2084.85,E2 -2084.85} C_VEL
LIN {X 0,Y 574.019,Z 382.437,A -85,B 0,C 180,E1 -2085.021,E2 -2085.021} C_VEL
LIN {X 0,Y 573.035,Z 377.464,A -85,B 0,C 180,E1 -2085.13,E2 -2085.13} C_VEL
LIN {X 0,Y 573.045,Z 371.497,A -85,B 0,C 180,E1 -2087.855,E2 -2087.855} C_VEL
LIN {X 0,Y 573.031,Z 366.683,A -85,B 0,C 180,E1 -2090.085,E2 -2090.085} C_VEL
LIN {X 0,Y 573.075,Z 361.87,A -85,B 0,C 180,E1 -2092.345,E2 -2092.345} C_VEL
LIN {X 0,Y 573.118,Z 355.463,A -85,B 0,C 180,E1 -2095.417,E2 -2095.417} C_VEL
LIN {X 0,Y 573.184,Z 350.28,A -85,B 0,C 180,E1 -2098.016,E2 -2098.016} C_VEL
LIN {X 0,Y 573.218,Z 344.668,A -85,B 0,C 180,E1 -2100.88,E2 -2100.88} C_VEL
LIN {X 0,Y 573.294,Z 339.581,A -85,B 0,C 180,E1 -2103.528,E2 -2103.528} C_VEL
LIN {X 0,Y 573.35,Z 334.853,A -85,B 0,C 180,E1 -2106.042,E2 -2106.042} C_VEL
LIN {X 0,Y 573.28,Z 329.761,A -85,B 0,C 180,E1 -2108.755,E2 -2108.755} C_VEL
LIN {X 0,Y 573.236,Z 329.709,A -85,B 0,C 180,E1 -2111.593,E2 -2111.593} C_VEL
LIN {X 0,Y 573.241,Z 329.704,A -85,B 0,C 180,E1 -2114.334,E2 -2114.334} C_VEL
LIN {X 0,Y 573.245,Z 329.701,A -85,B 0,C 180,E1 -2117.359,E2 -2117.359} C_VEL
LIN {X 0,Y 573.246,Z 329.702,A -85,B 0,C 180,E1 -2120.393,E2 -2120.393} C_VEL
LIN {X 0,Y 573.257,Z 329.705,A -85,B 0,C 180,E1 -2123.078,E2 -2123.078} C_VEL
LIN {X 0,Y 573.273,Z 329.698,A -85,B 0,C 180,E1 -2125.672,E2 -2125.672} C_VEL
LIN {X 0,Y 573.245,Z 329.708,A -85,B 0,C 180,E1 -2128.185,E2 -2128.185} C_VEL
LIN {X 0,Y 573.27,Z 329.698,A -85,B 0,C 180,E1 -2130.634,E2 -2130.634} C_VEL
LIN {X 0,Y 573.256,Z 329.704,A -85,B 0,C 180,E1 -2133.024,E2 -2133.024} C_VEL
LIN {X 0,Y 573.281,Z 329.699,A -85,B 0,C 180,E1 -2135.366,E2 -2135.366} C_VEL
LIN {X 0,Y 573.235,Z 329.708,A -85,B 0,C 180,E1 -2138.419,E2 -2138.419} C_VEL
LIN {X 0,Y 573.276,Z 329.698,A -85,B 0,C 180,E1 -2140.731,E2 -2140.731} C_VEL
LIN {X 0,Y 573.258,Z 329.703,A -85,B 0,C 180,E1 -2143.622,E2 -2143.622} C_VEL
LIN {X 0,Y 573.273,Z 329.698,A -85,B 0,C 180,E1 -2145.807,E2 -2145.807} C_VEL
LIN {X 0,Y 573.27,Z 329.701,A -85,B 0,C 180,E1 -2148.745,E2 -2148.745} C_VEL
LIN {X 0,Y 573.261,Z 329.703,A -85,B 0,C 180,E1 -2151.54,E2 -2151.54} C_VEL
LIN {X 0,Y 573.247,Z 329.705,A -85,B 0,C 180,E1 -2153.665,E2 -2153.665} C_VEL
LIN {X 0,Y 573.226,Z 329.704,A -85,B 0,C 180,E1 -2155.781,E2 -2155.781} C_VEL
LIN {X 0,Y 573.307,Z 329.694,A -85,B 0,C 180,E1 -2157.892,E2 -2157.892} C_VEL
LIN {X 0,Y 573.336,Z 329.69,A -85,B 0,C 180,E1 -2160.702,E2 -2160.702} C_VEL
LIN {X 0,Y 573.31,Z 329.693,A -85,B 0,C 180,E1 -2162.81,E2 -2162.81} C_VEL
LIN {X 0,Y 573.295,Z 329.697,A -85,B 0,C 180,E1 -2165.628,E2 -2165.628} C_VEL
LIN {X 0,Y 573.278,Z 329.697,A -85,B 0,C 180,E1 -2167.75,E2 -2167.75} C_VEL
LIN {X 0,Y 573.269,Z 329.7,A -85,B 0,C 180,E1 -2170.596,E2 -2170.596} C_VEL
LIN {X 0,Y 573.271,Z 329.699,A -85,B 0,C 180,E1 -2172.748,E2 -2172.748} C_VEL
LIN {X 0,Y 573.24,Z 329.705,A -85,B 0,C 180,E1 -2174.919,E2 -2174.919} C_VEL
LIN {X 0,Y 573.25,Z 329.701,A -85,B 0,C 180,E1 -2177.848,E2 -2177.848} C_VEL
LIN {X 0,Y 573.247,Z 329.705,A -85,B 0,C 180,E1 -2180.077,E2 -2180.077} C_VEL
LIN {X 0,Y 573.241,Z 329.704,A -85,B 0,C 180,E1 -2182.338,E2 -2182.338} C_VEL
LIN {X 0,Y 573.259,Z 329.706,A -85,B 0,C 180,E1 -2185.41,E2 -2185.41} C_VEL
LIN {X 0,Y 573.257,Z 329.7,A -85,B 0,C 180,E1 -2188.029,E2 -2188.029} C_VEL
LIN {X 0,Y 573.251,Z 329.705,A -85,B 0,C 180,E1 -2190.176,E2 -2190.176} C_VEL
LIN {X 0,Y 573.256,Z 329.701,A -85,B 0,C 180,E1 -2192.645,E2 -2192.645} C_VEL
LIN {X 0,Y 573.271,Z 329.703,A -85,B 0,C 180,E1 -2195.183,E2 -2195.183} C_VEL
LIN {X 0,Y 573.24,Z 329.703,A -85,B 0,C 180,E1 -2197.807,E2 -2197.807} C_VEL
LIN {X 0,Y 573.248,Z 329.708,A -85,B 0,C 180,E1 -2200.525,E2 -2200.525} C_VEL
LIN {X 0,Y 573.239,Z 329.705,A -85,B 0,C 180,E1 -2203.359,E2 -2203.359} C_VEL
LIN {X 0,Y 573.257,Z 329.701,A -85,B 0,C 180,E1 -2206.33,E2 -2206.33} C_VEL
LIN {X 0,Y 573.247,Z 329.705,A -85,B 0,C 180,E1 -2208.544,E2 -2208.544} C_VEL
LIN {X 0,Y 573.245,Z 329.704,A -85,B 0,C 180,E1 -2211.298,E2 -2211.298} C_VEL
LIN {X 0,Y 573.267,Z 329.715,A -85,B 0,C 180,E1 -2213.734,E2 -2213.734} C_VEL
LIN {X 0,Y 574.003,Z 334.228,A -85,B 0,C 180,E1 -2215.118,E2 -2215.118} C_VEL
LIN {X 0,Y 573.891,Z 342.267,A -85,B 0,C 180,E1 -2217.395,E2 -2217.395} C_VEL
LIN {X 0,Y 573.757,Z 352.512,A -85,B 0,C 180,E1 -2220.182,E2 -2220.182} C_VEL
LIN {X 0,Y 573.619,Z 363.339,A -85,B 0,C 180,E1 -2223.042,E2 -2223.042} C_VEL
LIN {X 0,Y 573.505,Z 373.873,A -85,B 0,C 180,E1 -2225.762,E2 -2225.762} C_VEL
LIN {X 0,Y 573.405,Z 384.407,A -85,B 0,C 180,E1 -2228.426,E2 -2228.426} C_VEL
LIN {X 0,Y 573.269,Z 396.446,A -85,B 0,C 180,E1 -2231.413,E2 -2231.413} C_VEL
LIN {X 0,Y 573.271,Z 400.457,A -85,B 0,C 180,E1 -2232.366,E2 -2232.366} C_VEL
LIN {X 0,Y 574.762,Z 407.3,A -85,B 0,C 180,E1 -2232.507,E2 -2232.507} C_VEL
LIN {X 0,Y 574.652,Z 422.474,A -85,B 0,C 180,E1 -2232.799,E2 -2232.799} C_VEL
LIN {X 0,Y 574.512,Z 437.902,A -85,B 0,C 180,E1 -2233.247,E2 -2233.247} C_VEL
LIN {X 0,Y 574.278,Z 452.817,A -85,B 0,C 180,E1 -2233.834,E2 -2233.834} C_VEL
LIN {X 0,Y 574.088,Z 467.098,A -85,B 0,C 180,E1 -2234.558,E2 -2234.558} C_VEL
LIN {X 0,Y 573.891,Z 480.684,A -85,B 0,C 180,E1 -2235.411,E2 -2235.411} C_VEL
LIN {X 0,Y 573.689,Z 493.161,A -85,B 0,C 180,E1 -2236.36,E2 -2236.36} C_VEL
LIN {X 0,Y 573.511,Z 504.969,A -85,B 0,C 180,E1 -2237.437,E2 -2237.437} C_VEL
LIN {X 0,Y 573.349,Z 514.9,A -85,B 0,C 180,E1 -2238.51,E2 -2238.51} C_VEL
LIN {X 0,Y 573.256,Z 524.618,A -85,B 0,C 180,E1 -2239.76,E2 -2239.76} C_VEL
LIN {X 0,Y 573.135,Z 532.72,A -85,B 0,C 180,E1 -2241.005,E2 -2241.005} C_VEL
LIN {X 0,Y 573.093,Z 539.424,A -85,B 0,C 180,E1 -2242.247,E2 -2242.247} C_VEL
LIN {X 0,Y 573.015,Z 545.606,A -85,B 0,C 180,E1 -2243.662,E2 -2243.662} C_VEL
LIN {X 0,Y 572.951,Z 550.384,A -85,B 0,C 180,E1 -2245.074,E2 -2245.074} C_VEL
LIN {X 0,Y 573.004,Z 553.888,A -85,B 0,C 180,E1 -2246.484,E2 -2246.484} C_VEL
LIN {X 0,Y 572.938,Z 556.192,A -85,B 0,C 180,E1 -2247.891,E2 -2247.891} C_VEL
LIN {X 0,Y 572.938,Z 557.349,A -85,B 0,C 180,E1 -2249.297,E2 -2249.297} C_VEL
LIN {X 0,Y 572.938,Z 557.349,A -85,B 0,C 180,E1 -2250.703,E2 -2250.703} C_VEL
LIN {X 0,Y 572.938,Z 556.191,A -85,B 0,C 180,E1 -2252.109,E2 -2252.109} C_VEL
LIN {X 0,Y 573.004,Z 553.887,A -85,B 0,C 180,E1 -2253.516,E2 -2253.516} C_VEL
LIN {X 0,Y 572.951,Z 550.385,A -85,B 0,C 180,E1 -2254.926,E2 -2254.926} C_VEL
LIN {X 0,Y 573.014,Z 545.608,A -85,B 0,C 180,E1 -2256.337,E2 -2256.337} C_VEL
LIN {X 0,Y 573.093,Z 539.423,A -85,B 0,C 180,E1 -2257.753,E2 -2257.753} C_VEL
LIN {X 0,Y 573.135,Z 531.649,A -85,B 0,C 180,E1 -2259.173,E2 -2259.173} C_VEL
LIN {X 0,Y 573.27,Z 523.369,A -85,B 0,C 180,E1 -2260.418,E2 -2260.418} C_VEL
LIN {X 0,Y 573.386,Z 513.391,A -85,B 0,C 180,E1 -2261.668,E2 -2261.668} C_VEL
LIN {X 0,Y 573.568,Z 503.189,A -85,B 0,C 180,E1 -2262.742,E2 -2262.742} C_VEL
LIN {X 0,Y 573.705,Z 491.018,A -85,B 0,C 180,E1 -2263.82,E2 -2263.82} C_VEL
LIN {X 0,Y 573.963,Z 477.901,A -85,B 0,C 180,E1 -2264.781,E2 -2264.781} C_VEL
LIN {X 0,Y 574.136,Z 465.516,A -85,B 0,C 180,E1 -2265.532,E2 -2265.532} C_VEL
LIN {X 0,Y 574.326,Z 450.832,A -85,B 0,C 180,E1 -2266.256,E2 -2266.256} C_VEL
LIN {X 0,Y 574.52,Z 436.613,A -85,B 0,C 180,E1 -2266.798,E2 -2266.798} C_VEL
LIN {X 0,Y 574.661,Z 421.78,A -85,B 0,C 180,E1 -2267.218,E2 -2267.218} C_VEL
LIN {X 0,Y 574.658,Z 406.609,A -85,B 0,C 180,E1 -2267.506,E2 -2267.506} C_VEL
LIN {X 0,Y 573.278,Z 400.274,A -85,B 0,C 180,E1 -2267.647,E2 -2267.647} C_VEL
LIN {X 0,Y 573.342,Z 388.922,A -85,B 0,C 180,E1 -2270.448,E2 -2270.448} C_VEL
LIN {X 0,Y 573.492,Z 376.841,A -85,B 0,C 180,E1 -2273.481,E2 -2273.481} C_VEL
LIN {X 0,Y 573.601,Z 364.844,A -85,B 0,C 180,E1 -2276.565,E2 -2276.565} C_VEL
LIN {X 0,Y 573.734,Z 353.36,A -85,B 0,C 180,E1 -2279.574,E2 -2279.574} C_VEL
LIN {X 0,Y 573.919,Z 343.233,A -85,B 0,C 180,E1 -2282.334,E2 -2282.334} C_VEL
LIN {X 0,Y 574.014,Z 335.287,A -85,B 0,C 180,E1 -2284.579,E2 -2284.579} C_VEL
LIN {X 0,Y 573.651,Z 331.94,A -85,B 0,C 180,E1 -2285.573,E2 -2285.573} C_VEL
LIN {X 0,Y 573.251,Z 329.708,A -85,B 0,C 180,E1 -2286.321,E2 -2286.321} C_VEL
LIN {X 0,Y 573.244,Z 329.704,A -85,B 0,C 180,E1 -2288.702,E2 -2288.702} C_VEL
LIN {X 0,Y 573.256,Z 329.702,A -85,B 0,C 180,E1 -2291.596,E2 -2291.596} C_VEL
LIN {X 0,Y 573.24,Z 329.706,A -85,B 0,C 180,E1 -2294.333,E2 -2294.333} C_VEL
LIN {X 0,Y 573.242,Z 329.704,A -85,B 0,C 180,E1 -2297.359,E2 -2297.359} C_VEL
LIN {X 0,Y 573.251,Z 329.701,A -85,B 0,C 180,E1 -2300.393,E2 -2300.393} C_VEL
LIN {X 0,Y 573.26,Z 329.705,A -85,B 0,C 180,E1 -2303.078,E2 -2303.078} C_VEL
LIN {X 0,Y 573.276,Z 329.699,A -85,B 0,C 180,E1 -2305.672,E2 -2305.672} C_VEL
LIN {X 0,Y 573.242,Z 329.706,A -85,B 0,C 180,E1 -2308.185,E2 -2308.185} C_VEL
LIN {X 0,Y 573.268,Z 329.699,A -85,B 0,C 180,E1 -2310.634,E2 -2310.634} C_VEL
LIN {X 0,Y 573.255,Z 329.707,A -85,B 0,C 180,E1 -2313.024,E2 -2313.024} C_VEL
LIN {X 0,Y 573.28,Z 329.697,A -85,B 0,C 180,E1 -2315.366,E2 -2315.366} C_VEL
LIN {X 0,Y 573.233,Z 329.704,A -85,B 0,C 180,E1 -2318.42,E2 -2318.42} C_VEL
LIN {X 0,Y 573.274,Z 329.698,A -85,B 0,C 180,E1 -2320.731,E2 -2320.731} C_VEL
LIN {X 0,Y 573.255,Z 329.7,A -85,B 0,C 180,E1 -2323.622,E2 -2323.622} C_VEL
